C01810=1051.567,302.793,393.168,172.665,38.135,157.229
C01811=1051.561,302.545,393.201,172.661,38.131,157.228
C01812=1051.554,302.298,393.234,172.658,38.128,157.227
C01813=1051.547,302.050,393.266,172.655,38.124,157.226
C01814=1051.541,301.803,393.299,172.651,38.120,157.225
C01815=1051.534,301.555,393.332,172.648,38.117,157.225
C01816=1051.528,301.307,393.364,172.644,38.114,157.224
C01817=1051.521,301.059,393.397,172.641,38.110,157.223
C01818=1051.515,300.812,393.430,172.638,38.106,157.222
C01819=1051.508,300.565,393.462,172.634,38.103,157.221
C01820=1051.501,300.316,393.495,172.631,38.099,157.220
C01821=1051.495,300.069,393.528,172.628,38.096,157.220
C01822=1051.489,299.820,393.560,172.624,38.093,157.219
C01823=1051.483,299.573,393.593,172.621,38.089,157.218
C01824=1051.476,299.326,393.625,172.618,38.085,157.217
C01825=1051.469,299.078,393.658,172.614,38.082,157.216
C01826=1051.463,298.830,393.690,172.611,38.078,157.215
C01827=1051.457,298.582,393.722,172.608,38.075,157.215
C01828=1051.450,298.334,393.755,172.604,38.072,157.214
C01829=1051.443,298.087,393.788,172.601,38.068,157.213
C01830=1051.437,297.838,393.820,172.598,38.065,157.212
C01831=1051.431,297.591,393.852,172.595,38.061,157.211
C01832=1051.425,297.343,393.885,172.591,38.057,157.210
C01833=1051.419,297.095,393.917,172.587,38.054,157.210
C01834=1051.412,296.848,393.949,172.585,38.051,157.209
C01835=1051.405,296.600,393.982,172.581,38.047,157.208
C01836=1051.399,296.352,394.014,172.578,38.044,157.207
C01837=1051.392,296.105,394.046,172.575,38.040,157.206
C01838=1051.386,295.856,394.078,172.571,38.037,157.205
C01839=1051.379,295.609,394.110,172.569,38.033,157.205
C01840=1051.373,295.361,394.142,172.565,38.030,157.204
C01841=1051.366,295.114,394.175,172.561,38.027,157.203
C01842=1051.360,294.865,394.207,172.559,38.023,157.202
C01843=1051.353,294.617,394.239,172.555,38.020,157.201
C01844=1051.347,294.369,394.271,172.552,38.016,157.201
C01845=1051.340,294.122,394.303,172.549,38.013,157.200
C01846=1051.334,293.874,394.335,172.545,38.010,157.199
C01847=1051.327,293.626,394.367,172.542,38.006,157.198
C01848=1051.320,293.379,394.399,172.539,38.003,157.197
C01849=1051.314,293.130,394.431,172.536,37.999,157.197
C01850=1051.307,292.882,394.462,172.533,37.996,157.196
C01851=1051.300,292.635,394.494,172.529,37.993,157.195
C01852=1051.294,292.387,394.526,172.526,37.990,157.194
C01853=1051.287,292.139,394.558,172.523,37.986,157.193
C01854=1051.281,291.891,394.590,172.520,37.983,157.193
C01855=1051.274,291.644,394.622,172.516,37.979,157.192
C01856=1051.268,291.396,394.654,172.513,37.976,157.191
C01857=1051.262,291.147,394.686,172.510,37.972,157.190
C01858=1051.255,290.882,394.720,172.506,37.969,157.189
C01859=1051.247,290.617,394.753,172.503,37.966,157.189
C01860=1051.240,290.351,394.787,172.500,37.962,157.188
C01861=1051.233,290.085,394.821,172.496,37.958,157.187
C01862=1051.226,289.838,394.853,172.493,37.955,157.186
C01863=1051.220,289.589,394.885,172.490,37.952,157.185
C01864=1051.213,289.341,394.917,172.487,37.949,157.185
C01865=1051.207,289.094,394.948,172.484,37.945,157.184
C01866=1051.201,288.846,394.980,172.480,37.942,157.183
C01867=1051.195,288.598,395.011,172.478,37.938,157.182
C01868=1051.188,288.350,395.043,172.474,37.935,157.181
C01869=1051.181,288.102,395.074,172.471,37.932,157.181
C01870=1051.175,287.854,395.106,172.468,37.929,157.180
C01871=1051.168,287.606,395.138,172.465,37.925,157.179
C01872=1051.162,287.358,395.169,172.462,37.922,157.178
C01873=1051.155,287.110,395.200,172.459,37.919,157.178
C01874=1051.148,286.863,395.232,172.455,37.915,157.177
C01875=1051.142,286.615,395.263,172.453,37.912,157.176
C01876=1051.135,286.367,395.294,172.449,37.909,157.175
C01877=1051.129,286.120,395.326,172.447,37.906,157.175
C01878=1051.122,285.871,395.356,172.443,37.902,157.174
C01879=1051.116,285.623,395.388,172.440,37.899,157.173
C01880=1051.109,285.375,395.419,172.437,37.896,157.172
C01881=1051.102,285.127,395.451,172.434,37.892,157.171
C01882=1051.095,284.879,395.482,172.431,37.889,157.171
C01883=1051.089,284.632,395.514,172.428,37.886,157.170
C01884=1051.083,284.384,395.544,172.424,37.883,157.169
C01885=1051.076,284.136,395.575,172.422,37.879,157.168
C01886=1051.069,283.888,395.607,172.418,37.876,157.168
C01887=1051.063,283.640,395.639,172.416,37.873,157.167
C01888=1051.057,283.391,395.670,172.412,37.870,157.166
C01889=1051.051,283.144,395.701,172.409,37.866,157.165
C01890=1051.044,282.896,395.732,172.406,37.863,157.165
C01891=1051.038,282.648,395.763,172.403,37.860,157.164
C01892=1051.031,282.400,395.794,172.401,37.856,157.163
C01893=1051.024,282.152,395.826,172.397,37.853,157.162
C01894=1051.018,281.904,395.856,172.394,37.850,157.162
C01895=1051.012,281.656,395.887,172.391,37.847,157.161
C01896=1051.005,281.408,395.919,172.388,37.844,157.160
C01897=1050.999,281.160,395.950,172.385,37.840,157.159
C01898=1050.992,280.912,395.981,172.382,37.837,157.159
C01899=1050.986,280.664,396.011,172.379,37.833,157.158
C01900=1050.979,280.416,396.043,172.376,37.830,157.157
C01901=1050.973,280.169,396.074,172.373,37.827,157.156
C01902=1050.967,279.920,396.105,172.370,37.824,157.155
C01903=1050.960,279.672,396.136,172.367,37.821,157.155
C01904=1050.954,279.424,396.166,172.365,37.817,157.154
C01905=1050.947,279.177,396.197,172.361,37.814,157.153
C01906=1050.940,278.928,396.228,172.358,37.811,157.153
C01907=1050.934,278.680,396.259,172.355,37.807,157.152
C01908=1050.928,278.433,396.290,172.352,37.805,157.151
C01909=1050.921,278.184,396.320,172.349,37.801,157.150
C01910=1050.914,277.937,396.351,172.346,37.798,157.150
C01911=1050.908,277.689,396.382,172.344,37.795,157.149
C01912=1050.902,277.440,396.412,172.340,37.791,157.148
C01913=1050.895,277.192,396.444,172.337,37.788,157.147
C01914=1050.889,276.938,396.475,172.335,37.785,157.147
C01915=1050.882,276.684,396.507,172.331,37.782,157.146
C01916=1050.875,276.430,396.538,172.329,37.779,157.145
C01917=1050.868,276.175,396.569,172.325,37.775,157.144
C01918=1050.862,275.927,396.600,172.322,37.772,157.144
C01919=1050.855,275.679,396.630,172.320,37.769,157.143
C01920=1050.849,275.432,396.661,172.316,37.765,157.142
C01921=1050.843,275.184,396.692,172.314,37.762,157.141
C01922=1050.836,274.935,396.722,172.310,37.759,157.141
C01923=1050.830,274.688,396.752,172.308,37.756,157.140
C01924=1050.823,274.439,396.783,172.305,37.753,157.139
C01925=1050.816,274.191,396.814,172.302,37.750,157.138
C01926=1050.810,273.944,396.844,172.299,37.746,157.138
C01927=1050.803,273.695,396.875,172.296,37.743,157.137
C01928=1050.798,273.447,396.905,172.293,37.740,157.136
C01929=1050.791,273.199,396.935,172.290,37.737,157.135
C01930=1050.785,272.951,396.966,172.288,37.734,157.135
C01931=1050.778,272.703,396.996,172.284,37.730,157.134
C01932=1050.771,272.454,397.026,172.282,37.727,157.133
C01933=1050.765,272.207,397.057,172.279,37.724,157.133
C01934=1050.759,271.959,397.088,172.276,37.721,157.132
C01935=1050.752,271.711,397.118,172.273,37.717,157.131
C01936=1050.746,271.463,397.149,172.270,37.715,157.130
C01937=1050.739,271.215,397.178,172.268,37.711,157.130
C01938=1050.733,270.967,397.209,172.264,37.708,157.129
C01939=1050.726,270.719,397.238,172.262,37.705,157.128
C01940=1050.720,270.470,397.269,172.259,37.702,157.128
C01941=1050.713,270.222,397.299,172.256,37.698,157.127
C01942=1050.707,269.974,397.329,172.253,37.695,157.126
C01943=1050.700,269.726,397.360,172.250,37.692,157.125
C01944=1050.694,269.478,397.390,172.248,37.689,157.125
C01945=1050.687,269.230,397.420,172.244,37.686,157.124
C01946=1050.681,268.982,397.450,172.242,37.683,157.123
C01947=1050.674,268.734,397.480,172.239,37.680,157.123
C01948=1050.668,268.486,397.511,172.237,37.676,157.122
C01949=1050.662,268.238,397.540,172.233,37.673,157.121
C01950=1050.655,267.989,397.571,172.231,37.670,157.120
C01951=1050.649,267.742,397.600,172.228,37.667,157.120
C01952=1050.642,267.493,397.630,172.225,37.664,157.119
C01953=1050.636,267.245,397.660,172.222,37.661,157.118
C01954=1050.629,266.997,397.690,172.220,37.658,157.117
C01955=1050.622,266.749,397.720,172.217,37.654,157.117
C01956=1050.616,266.501,397.751,172.213,37.651,157.116
C01957=1050.610,266.253,397.780,172.211,37.648,157.115
C01958=1050.603,266.004,397.810,172.208,37.645,157.115
C01959=1050.597,265.757,397.840,172.206,37.642,157.114
C01960=1050.590,265.508,397.870,172.203,37.639,157.113
C01961=1050.584,265.260,397.900,172.200,37.636,157.112
C01962=1050.578,265.012,397.930,172.197,37.632,157.112
C01963=1050.571,264.764,397.959,172.195,37.629,157.111
C01964=1050.565,264.516,397.989,172.192,37.626,157.110
C01965=1050.558,264.268,398.020,172.189,37.623,157.110
C01966=1050.552,264.019,398.049,172.186,37.619,157.109
C01967=1050.546,263.772,398.079,172.183,37.617,157.108
C01968=1050.539,263.523,398.108,172.181,37.614,157.108
C01969=1050.532,263.275,398.138,172.178,37.610,157.107
C01970=1050.526,263.025,398.168,172.175,37.607,157.106
C01971=1050.520,262.776,398.198,172.172,37.604,157.105
C01972=1050.513,262.526,398.228,172.170,37.601,157.105
C01973=1050.507,262.275,398.258,172.167,37.598,157.104
C01974=1050.500,262.026,398.287,172.165,37.594,157.103
C01975=1050.493,261.779,398.317,172.161,37.592,157.103
C01976=1050.487,261.531,398.346,172.159,37.589,157.102
C01977=1050.479,261.283,398.376,172.156,37.586,157.101
C01978=1050.473,261.035,398.405,172.154,37.582,157.100
C01979=1050.466,260.786,398.434,172.150,37.579,157.100
C01980=1050.459,260.538,398.464,172.148,37.576,157.099
C01981=1050.453,260.290,398.493,172.145,37.573,157.098
C01982=1050.446,260.041,398.522,172.143,37.570,157.098
C01983=1050.440,259.794,398.552,172.140,37.567,157.097
C01984=1050.434,259.546,398.581,172.138,37.564,157.096
C01985=1050.427,259.297,398.610,172.134,37.561,157.096
C01986=1050.420,259.049,398.639,172.132,37.558,157.095
C01987=1050.414,258.801,398.669,172.129,37.555,157.094
C01988=1050.407,258.553,398.699,172.127,37.552,157.094
C01989=1050.401,258.304,398.728,172.124,37.548,157.093
C01990=1050.395,258.056,398.757,172.122,37.546,157.092
C01991=1050.387,257.808,398.787,172.118,37.543,157.092
C01992=1050.381,257.560,398.816,172.115,37.539,157.091
C01993=1050.375,257.312,398.845,172.113,37.536,157.090
C01994=1050.368,257.063,398.874,172.111,37.533,157.089
C01995=1050.362,256.815,398.903,172.108,37.530,157.089
C01996=1050.356,256.567,398.932,172.105,37.527,157.088
C01997=1050.349,256.319,398.962,172.103,37.524,157.087
C01998=1050.342,256.070,398.992,172.099,37.521,157.087
C01999=1050.336,255.822,399.021,172.097,37.518,157.086
C02000=1050.329,255.574,399.049,172.094,37.515,157.085
C02001=1050.323,255.326,399.078,172.092,37.512,157.085
C02002=1050.316,255.077,399.107,172.089,37.508,157.084
C02003=1050.310,254.829,399.136,172.087,37.505,157.083
C02004=1050.303,254.581,399.166,172.084,37.502,157.083
C02005=1050.297,254.333,399.195,172.082,37.499,157.082
C02006=1050.291,254.085,399.224,172.079,37.496,157.081
C02007=1050.284,253.836,399.253,172.077,37.493,157.080
C02008=1050.278,253.588,399.282,172.073,37.490,157.080
C02009=1050.271,253.340,399.311,172.071,37.487,157.079
C02010=1050.265,253.092,399.340,172.068,37.484,157.078
C02011=1050.258,252.844,399.369,172.066,37.480,157.078
C02012=1050.251,252.595,399.398,172.063,37.477,157.077
C02013=1050.245,252.347,399.427,172.061,37.474,157.076
C02014=1050.239,252.099,399.456,172.058,37.471,157.076
C02015=1050.233,251.851,399.485,172.056,37.468,157.075
C02016=1050.226,251.602,399.514,172.053,37.465,157.074
C02017=1050.220,251.354,399.543,172.051,37.461,157.073
C02018=1050.214,251.106,399.572,172.048,37.458,157.073
C02019=1050.208,250.858,399.601,172.046,37.456,157.072
C02020=1050.201,250.609,399.630,172.043,37.452,157.071
C02021=1050.194,250.361,399.658,172.041,37.449,157.071
C02022=1050.188,250.113,399.687,172.038,37.446,157.070
C02023=1050.182,249.865,399.716,172.036,37.443,157.069
C02024=1050.175,249.616,399.746,172.033,37.440,157.069
C02025=1050.169,249.368,399.775,172.031,37.437,157.068
C02026=1050.162,249.116,399.804,172.028,37.433,157.067
C02027=1050.156,248.865,399.833,172.026,37.430,157.067
C02028=1050.150,248.613,399.862,172.022,37.427,157.066
C02029=1050.144,248.362,399.891,172.020,37.424,157.065
C02030=1050.138,248.114,399.919,172.017,37.420,157.064
C02031=1050.131,247.865,399.948,172.015,37.417,157.064
C02032=1050.125,247.617,399.977,172.012,37.415,157.063
C02033=1050.119,247.369,400.007,172.010,37.411,157.062
C02034=1050.112,247.121,400.034,172.007,37.408,157.062
C02035=1050.106,246.873,400.063,172.005,37.405,157.061
C02036=1050.100,246.625,400.092,172.003,37.402,157.060
C02037=1050.094,246.376,400.121,172.001,37.399,157.060
C02038=1050.087,246.128,400.150,171.998,37.395,157.059
C02039=1050.081,245.879,400.179,171.996,37.392,157.058
C02040=1050.075,245.631,400.206,171.993,37.389,157.057
C02041=1050.068,245.382,400.236,171.991,37.386,157.057
C02042=1050.062,245.133,400.264,171.988,37.383,157.056
C02043=1050.055,244.886,400.293,171.986,37.380,157.055
C02044=1050.049,244.637,400.321,171.983,37.376,157.055
C02045=1050.042,244.389,400.349,171.981,37.373,157.054
C02046=1050.036,244.141,400.378,171.978,37.370,157.053
C02047=1050.030,243.892,400.407,171.976,37.367,157.053
C02048=1050.023,243.644,400.435,171.973,37.364,157.052
C02049=1050.017,243.396,400.464,171.971,37.361,157.051
C02050=1050.011,243.148,400.491,171.968,37.358,157.051
C02051=1050.004,242.900,400.520,171.966,37.355,157.050
C02052=1049.998,242.651,400.548,171.963,37.352,157.049
C02053=1049.991,242.403,400.577,171.961,37.349,157.049
C02054=1049.986,242.154,400.605,171.958,37.345,157.048
C02055=1049.979,241.907,400.633,171.956,37.342,157.047
C02056=1049.973,241.658,400.662,171.953,37.339,157.047
C02057=1049.966,241.409,400.690,171.951,37.336,157.046
C02058=1049.960,241.161,400.719,171.948,37.333,157.045
C02059=1049.953,240.913,400.746,171.946,37.330,157.044
C02060=1049.946,240.664,400.774,171.943,37.327,157.044
C02061=1049.940,240.416,400.803,171.942,37.323,157.043
C02062=1049.933,240.168,400.831,171.939,37.320,157.042
C02063=1049.927,239.919,400.859,171.937,37.317,157.042
C02064=1049.921,239.671,400.887,171.934,37.314,157.041
C02065=1049.914,239.423,400.915,171.932,37.311,157.040
C02066=1049.908,239.174,400.944,171.929,37.308,157.040
C02067=1049.901,238.926,400.971,171.927,37.305,157.039
C02068=1049.894,238.677,400.999,171.924,37.302,157.038
C02069=1049.888,238.429,401.028,171.922,37.299,157.038
C02070=1049.882,238.181,401.056,171.919,37.296,157.037
C02071=1049.875,237.933,401.083,171.917,37.293,157.036
C02072=1049.869,237.684,401.112,171.915,37.290,157.036
C02073=1049.863,237.436,401.139,171.913,37.286,157.035
C02074=1049.856,237.187,401.167,171.911,37.283,157.034
C02075=1049.849,236.939,401.195,171.908,37.280,157.034
C02076=1049.843,236.691,401.224,171.906,37.277,157.033
C02077=1049.837,236.442,401.252,171.903,37.274,157.032
C02078=1049.830,236.194,401.279,171.901,37.271,157.032
C02079=1049.824,235.946,401.307,171.898,37.268,157.031
C02080=1049.818,235.697,401.335,171.896,37.265,157.030
C02081=1049.811,235.449,401.363,171.893,37.261,157.030
C02082=1049.805,235.191,401.392,171.892,37.258,157.029
C02083=1049.797,234.934,401.421,171.889,37.255,157.028
C02084=1049.792,234.677,401.450,171.887,37.252,157.027
C02085=1049.784,234.419,401.478,171.884,37.248,157.027
C02086=1049.778,234.171,401.507,171.882,37.245,157.026
C02087=1049.772,233.922,401.534,171.879,37.242,157.025
C02088=1049.765,233.674,401.562,171.877,37.239,157.025
C02089=1049.759,233.426,401.589,171.874,37.236,157.024
C02090=1049.753,233.177,401.618,171.873,37.233,157.023
C02091=1049.746,232.929,401.645,171.870,37.230,157.023
C02092=1049.740,232.680,401.673,171.868,37.226,157.022
C02093=1049.733,232.432,401.701,171.865,37.224,157.021
C02094=1049.727,232.184,401.728,171.863,37.221,157.021
C02095=1049.721,231.935,401.756,171.860,37.217,157.020
C02096=1049.715,231.686,401.784,171.859,37.214,157.019
C02097=1049.708,231.438,401.811,171.857,37.211,157.019
C02098=1049.702,231.190,401.839,171.854,37.208,157.018
C02099=1049.695,230.942,401.866,171.852,37.205,157.017
C02100=1049.689,230.693,401.894,171.849,37.202,157.017
C02101=1049.682,230.445,401.922,171.847,37.199,157.016
C02102=1049.676,230.197,401.949,171.845,37.195,157.015
C02103=1049.669,229.948,401.976,171.843,37.192,157.015
C02104=1049.663,229.699,402.005,171.840,37.189,157.014
C02105=1049.657,229.451,402.032,171.838,37.186,157.013
C02106=1049.651,229.203,402.060,171.835,37.183,157.013
C02107=1049.644,228.954,402.087,171.834,37.180,157.012
C02108=1049.638,228.706,402.114,171.831,37.177,157.011
C02109=1049.631,228.457,402.142,171.829,37.173,157.010
C02110=1049.625,228.209,402.169,171.826,37.170,157.010
C02111=1049.618,227.961,402.196,171.824,37.167,157.009
C02112=1049.611,227.712,402.224,171.823,37.164,157.009
C02113=1049.605,227.463,402.251,171.820,37.161,157.008
C02114=1049.599,227.216,402.278,171.818,37.158,157.007
C02115=1049.592,226.967,402.306,171.815,37.155,157.007
C02116=1049.586,226.718,402.333,171.814,37.152,157.006
C02117=1049.579,226.470,402.361,171.811,37.148,157.005
C02118=1049.573,226.221,402.387,171.809,37.145,157.004
C02119=1049.566,225.973,402.415,171.806,37.142,157.004
C02120=1049.559,225.725,402.442,171.804,37.139,157.003
C02121=1049.553,225.476,402.469,171.802,37.136,157.002
C02122=1049.547,225.228,402.496,171.800,37.133,157.002
C02123=1049.540,224.979,402.523,171.797,37.130,157.001
C02124=1049.534,224.731,402.551,171.795,37.126,157.000
C02125=1049.528,224.482,402.578,171.794,37.123,157.000
C02126=1049.521,224.234,402.606,171.791,37.120,156.999
C02127=1049.515,223.985,402.632,171.789,37.117,156.999
C02128=1049.508,223.737,402.659,171.786,37.114,156.998
C02129=1049.502,223.489,402.686,171.785,37.111,156.997
C02130=1049.495,223.240,402.714,171.782,37.108,156.996
C02131=1049.489,222.991,402.741,171.780,37.104,156.996
C02132=1049.483,222.744,402.768,171.778,37.101,156.995
C02133=1049.477,222.494,402.795,171.776,37.098,156.994
C02134=1049.470,222.246,402.823,171.773,37.095,156.994
C02135=1049.463,221.998,402.849,171.771,37.092,156.993
C02136=1049.457,221.750,402.877,171.770,37.089,156.992
C02137=1049.451,221.501,402.903,171.767,37.085,156.992
C02138=1049.445,221.236,402.932,171.765,37.082,156.991
C02139=1049.437,220.971,402.961,171.762,37.079,156.990
C02140=1049.430,220.706,402.989,171.761,37.075,156.990
C02141=1049.424,220.441,403.019,171.758,37.072,156.989
C02142=1049.417,220.192,403.046,171.756,37.069,156.988
C02143=1049.411,219.944,403.072,171.753,37.066,156.987
C02144=1049.404,219.696,403.099,171.752,37.063,156.987
C02145=1049.398,219.447,403.126,171.749,37.059,156.986
C02146=1049.391,219.199,403.153,171.747,37.056,156.985
C02147=1049.385,218.950,403.180,171.744,37.053,156.985
C02148=1049.378,218.702,403.206,171.743,37.050,156.984
C02149=1049.371,218.453,403.233,171.740,37.047,156.983
C02150=1049.365,218.205,403.259,171.738,37.044,156.983
C02151=1049.359,217.956,403.286,171.737,37.041,156.982
C02152=1049.352,217.708,403.314,171.734,37.038,156.982
C02153=1049.345,217.460,403.340,171.732,37.034,156.981
C02154=1049.339,217.211,403.367,171.730,37.031,156.980
C02155=1049.333,216.962,403.393,171.728,37.028,156.979
C02156=1049.326,216.713,403.420,171.725,37.024,156.979
C02157=1049.320,216.465,403.447,171.724,37.021,156.978
C02158=1049.313,216.217,403.474,171.721,37.018,156.977
C02159=1049.307,215.969,403.501,171.719,37.015,156.977
C02160=1049.300,215.720,403.527,171.717,37.012,156.976
C02161=1049.294,215.471,403.554,171.715,37.009,156.975
C02162=1049.287,215.223,403.580,171.713,37.005,156.975
C02163=1049.281,214.974,403.607,171.711,37.002,156.974
C02164=1049.275,214.725,403.634,171.709,36.999,156.973
C02165=1049.269,214.477,403.660,171.707,36.996,156.973
C02166=1049.262,214.228,403.687,171.705,36.993,156.972
C02167=1049.256,213.980,403.713,171.702,36.989,156.971
C02168=1049.250,213.732,403.740,171.701,36.986,156.971
C02169=1049.243,213.483,403.766,171.698,36.983,156.970
C02170=1049.237,213.235,403.793,171.696,36.980,156.969
C02171=1049.230,212.986,403.819,171.695,36.977,156.969
C02172=1049.224,212.738,403.846,171.692,36.974,156.968
C02173=1049.217,212.489,403.872,171.691,36.970,156.967
C02174=1049.211,212.240,403.899,171.688,36.967,156.967
C02175=1049.204,211.992,403.925,171.686,36.964,156.966
C02176=1049.198,211.743,403.952,171.684,36.961,156.965
C02177=1049.192,211.495,403.978,171.682,36.958,156.965
C02178=1049.185,211.246,404.005,171.680,36.954,156.964
C02179=1049.179,210.998,404.031,171.678,36.951,156.963
C02180=1049.172,210.749,404.057,171.676,36.948,156.963
C02181=1049.166,210.501,404.084,171.674,36.944,156.962
C02182=1049.159,210.252,404.110,171.672,36.941,156.961
C02183=1049.153,210.004,404.137,171.670,36.938,156.960
C02184=1049.147,209.755,404.162,171.668,36.935,156.960
C02185=1049.140,209.507,404.189,171.665,36.932,156.959
C02186=1049.134,209.258,404.216,171.664,36.928,156.958
C02187=1049.127,209.009,404.242,171.661,36.925,156.958
C02188=1049.120,208.761,404.268,171.660,36.922,156.957
C02189=1049.114,208.513,404.293,171.657,36.919,156.956
C02190=1049.108,208.264,404.320,171.656,36.916,156.956
C02191=1049.101,208.016,404.346,171.654,36.912,156.955
C02192=1049.095,207.768,404.372,171.651,36.909,156.954
C02193=1049.088,207.518,404.399,171.650,36.906,156.954
C02194=1049.082,207.258,404.426,171.647,36.903,156.953
C02195=1049.075,207.000,404.453,171.646,36.899,156.952
C02196=1049.068,206.740,404.481,171.643,36.896,156.952
C02197=1049.061,206.481,404.508,171.641,36.892,156.951
C02198=1049.035,205.428,404.614,171.404,36.795,156.930
C02199=1049.029,205.180,404.639,171.402,36.792,156.929
C02200=1049.023,204.932,404.664,171.400,36.790,156.929
C02201=1049.017,204.683,404.689,171.396,36.788,156.928
C02202=1049.011,204.434,404.714,171.394,36.785,156.928
C02203=1049.005,204.185,404.739,171.392,36.783,156.927
C02204=1048.999,203.936,404.765,171.388,36.780,156.927
C02205=1048.993,203.688,404.789,171.386,36.778,156.926
C02206=1048.987,203.439,404.814,171.384,36.776,156.926
C02207=1048.981,203.190,404.839,171.382,36.773,156.925
C02208=1048.974,202.942,404.864,171.378,36.771,156.925
C02209=1048.969,202.694,404.888,171.376,36.768,156.924
C02210=1048.963,202.445,404.914,171.374,36.766,156.924
C02211=1048.957,202.196,404.938,171.370,36.763,156.923
C02212=1048.951,201.947,404.964,171.368,36.761,156.923
C02213=1048.945,201.699,404.989,171.366,36.759,156.923
C02214=1048.939,201.450,405.013,171.363,36.756,156.922
C02215=1048.932,201.201,405.038,171.360,36.754,156.922
C02216=1048.926,200.952,405.063,171.358,36.752,156.921
C02217=1048.921,200.704,405.088,171.355,36.750,156.921
C02218=1048.914,200.455,405.112,171.352,36.747,156.920
C02219=1048.908,200.206,405.137,171.350,36.745,156.920
C02220=1048.902,199.957,405.162,171.348,36.742,156.919
C02221=1048.895,199.709,405.186,171.345,36.741,156.919
C02222=1048.890,199.460,405.211,171.342,36.738,156.918
C02223=1048.883,199.211,405.235,171.340,36.736,156.918
C02224=1048.877,198.963,405.260,171.337,36.733,156.917
C02225=1048.871,198.714,405.284,171.335,36.731,156.917
C02226=1048.865,198.466,405.309,171.332,36.729,156.916
C02227=1048.859,198.216,405.334,171.329,36.727,156.916
C02228=1048.852,197.968,405.358,171.327,36.724,156.915
C02229=1048.847,197.719,405.383,171.325,36.722,156.915
C02230=1048.840,197.470,405.407,171.322,36.720,156.915
C02231=1048.834,197.222,405.432,171.319,36.718,156.914
C02232=1048.828,196.973,405.456,171.317,36.715,156.914
C02233=1048.822,196.724,405.480,171.315,36.713,156.913
C02234=1048.816,196.475,405.506,171.311,36.711,156.913
C02235=1048.809,196.227,405.529,171.309,36.709,156.912
C02236=1048.804,195.978,405.554,171.307,36.706,156.912
C02237=1048.797,195.729,405.578,171.305,36.704,156.911
C02238=1048.791,195.481,405.603,171.301,36.702,156.911
C02239=1048.785,195.232,405.627,171.299,36.700,156.910
C02240=1048.779,194.983,405.652,171.297,36.697,156.910
C02241=1048.774,194.734,405.676,171.294,36.695,156.909
C02242=1048.767,194.486,405.701,171.292,36.693,156.909
C02243=1048.761,194.237,405.725,171.289,36.690,156.908
C02244=1048.755,193.988,405.749,171.287,36.688,156.908
C02245=1048.749,193.739,405.773,171.284,36.686,156.908
C02246=1048.742,193.491,405.798,171.282,36.684,156.907
C02247=1048.736,193.242,405.822,171.279,36.681,156.907
C02248=1048.730,192.994,405.846,171.276,36.679,156.906
C02249=1048.725,192.744,405.871,171.274,36.677,156.906
C02250=1048.719,192.496,405.894,171.272,36.675,156.905
C02251=1048.713,192.247,405.919,171.270,36.672,156.905
C02252=1048.706,191.998,405.943,171.267,36.670,156.904
C02253=1048.700,191.750,405.968,171.264,36.668,156.904
C02254=1048.694,191.501,405.992,171.262,36.666,156.903
C02255=1048.688,191.252,406.016,171.259,36.663,156.903
C02256=1048.683,191.003,406.041,171.257,36.661,156.903
C02257=1048.676,190.755,406.065,171.255,36.659,156.902
C02258=1048.671,190.505,406.089,171.253,36.657,156.902
C02259=1048.664,190.221,406.116,171.249,36.654,156.901
C02260=1048.657,189.937,406.144,171.247,36.652,156.901
C02261=1048.650,189.652,406.172,171.244,36.649,156.900
C02262=1048.643,189.369,406.199,171.241,36.647,156.900
C02263=1048.637,189.119,406.224,171.239,36.644,156.899
C02264=1048.631,188.871,406.248,171.236,36.642,156.899
C02265=1048.625,188.622,406.272,171.233,36.640,156.898
C02266=1048.619,188.374,406.296,171.231,36.638,156.898
C02267=1048.613,188.124,406.321,171.229,36.635,156.897
C02268=1048.607,187.876,406.344,171.227,36.633,156.897
C02269=1048.602,187.627,406.368,171.224,36.631,156.896
C02270=1048.596,187.378,406.392,171.222,36.629,156.896
C02271=1048.590,187.129,406.416,171.219,36.627,156.896
C02272=1048.584,186.880,406.440,171.217,36.624,156.895
C02273=1048.578,186.632,406.464,171.214,36.622,156.895
C02274=1048.572,186.383,406.488,171.212,36.620,156.894
C02275=1048.566,186.134,406.513,171.210,36.618,156.894
C02276=1048.560,185.886,406.536,171.207,36.615,156.893
C02277=1048.554,185.637,406.560,171.205,36.613,156.893
C02278=1048.548,185.388,406.585,171.203,36.611,156.892
C02279=1048.543,185.139,406.607,171.201,36.609,156.892
C02280=1048.537,184.890,406.632,171.197,36.607,156.891
C02281=1048.531,184.642,406.656,171.195,36.604,156.891
C02282=1048.525,184.393,406.680,171.193,36.602,156.890
C02283=1048.519,184.144,406.704,171.190,36.600,156.890
C02284=1048.514,183.895,406.728,171.188,36.598,156.890
C02285=1048.507,183.646,406.752,171.186,36.596,156.889
C02286=1048.501,183.398,406.775,171.184,36.594,156.889
C02287=1048.494,183.148,406.798,171.181,36.592,156.888
C02288=1048.488,182.900,406.822,171.179,36.590,156.888
C02289=1048.481,182.651,406.846,171.176,36.587,156.888
C02290=1048.476,182.402,406.869,171.174,36.585,156.887
C02291=1048.469,182.153,406.893,171.171,36.584,156.887
C02292=1048.463,181.904,406.916,171.169,36.581,156.886
C02293=1048.457,181.656,406.939,171.167,36.579,156.886
C02294=1048.451,181.407,406.963,171.165,36.578,156.886
C02295=1048.445,181.158,406.986,171.162,36.575,156.885
C02296=1048.438,180.909,407.010,171.160,36.573,156.885
C02297=1048.432,180.660,407.033,171.157,36.571,156.884
C02298=1048.426,180.411,407.057,171.155,36.570,156.884
C02299=1048.420,180.163,407.080,171.152,36.567,156.883
C02300=1048.414,179.914,407.104,171.150,36.565,156.883
C02301=1048.408,179.665,407.127,171.148,36.564,156.883
C02302=1048.401,179.417,407.150,171.146,36.561,156.882
C02303=1048.395,179.168,407.173,171.144,36.559,156.882
C02304=1048.389,178.919,407.197,171.141,36.557,156.882
C02305=1048.383,178.670,407.220,171.139,36.555,156.881
C02306=1048.376,178.421,407.244,171.137,36.553,156.881
C02307=1048.371,178.172,407.267,171.134,36.551,156.880
C02308=1048.364,177.924,407.291,171.131,36.549,156.880
C02309=1048.358,177.674,407.314,171.129,36.547,156.879
C02310=1048.352,177.426,407.338,171.127,36.545,156.879
C02311=1048.346,177.177,407.361,171.125,36.543,156.879
C02312=1048.340,176.927,407.384,171.122,36.541,156.878
C02313=1048.333,176.679,407.407,171.120,36.539,156.878
C02314=1048.328,176.431,407.430,171.118,36.537,156.877
C02315=1048.321,176.182,407.454,171.116,36.535,156.877
C02316=1048.315,175.933,407.477,171.113,36.533,156.877
C02317=1048.309,175.684,407.500,171.111,36.531,156.876
C02318=1048.303,175.436,407.524,171.109,36.529,156.876
C02319=1048.297,175.186,407.547,171.107,36.527,156.875
C02320=1048.291,174.937,407.570,171.104,36.525,156.875
C02321=1048.285,174.689,407.593,171.102,36.523,156.875
C02322=1048.279,174.440,407.616,171.100,36.521,156.874
C02323=1048.272,174.155,407.643,171.097,36.518,156.874
C02324=1048.264,173.870,407.669,171.094,36.517,156.873
C02325=1048.258,173.585,407.696,171.092,36.514,156.873
C02326=1048.251,173.300,407.722,171.089,36.512,156.872
C02327=1048.245,173.052,407.745,171.087,36.510,156.872
C02328=1048.239,172.803,407.768,171.084,36.508,156.872
C02329=1048.233,172.554,407.791,171.082,36.506,156.871
C02330=1048.227,172.305,407.814,171.080,36.504,156.871
C02331=1048.221,172.056,407.838,171.078,36.502,156.870
C02332=1048.215,171.807,407.861,171.075,36.499,156.870
C02333=1048.209,171.558,407.884,171.073,36.498,156.870
C02334=1048.203,171.310,407.906,171.071,36.496,156.869
C02335=1048.197,171.060,407.930,171.069,36.494,156.869
C02336=1048.190,170.812,407.953,171.066,36.492,156.868
C02337=1048.185,170.563,407.976,171.064,36.490,156.868
C02338=1048.179,170.314,407.999,171.062,36.488,156.868
C02339=1048.173,170.065,408.022,171.060,36.485,156.867
C02340=1048.167,169.817,408.045,171.057,36.484,156.867
C02341=1048.161,169.568,408.067,171.055,36.482,156.866
C02342=1048.155,169.318,408.091,171.053,36.480,156.866
C02343=1048.149,169.069,408.114,171.051,36.477,156.866
C02344=1048.143,168.821,408.137,171.049,36.476,156.865
C02345=1048.137,168.572,408.160,171.046,36.474,156.865
C02346=1048.131,168.324,408.183,171.044,36.472,156.864
C02347=1048.125,168.075,408.206,171.042,36.470,156.864
C02348=1048.119,167.826,408.229,171.040,36.468,156.864
C02349=1048.114,167.577,408.252,171.037,36.466,156.863
C02350=1048.108,167.328,408.274,171.035,36.463,156.863
C02351=1048.102,167.078,408.298,171.033,36.462,156.862
C02352=1048.095,166.830,408.320,171.031,36.460,156.862
C02353=1048.089,166.581,408.343,171.028,36.458,156.862
C02354=1048.084,166.332,408.366,171.026,36.455,156.861
C02355=1048.078,166.083,408.389,171.025,36.454,156.861
C02356=1048.072,165.834,408.412,171.023,36.452,156.860
C02357=1048.066,165.586,408.434,171.021,36.450,156.860
C02358=1048.060,165.337,408.457,171.018,36.447,156.860
C02359=1048.054,165.088,408.480,171.016,36.446,156.859
C02360=1048.048,164.839,408.503,171.014,36.444,156.859
C02361=1048.043,164.590,408.526,171.012,36.442,156.858
C02362=1048.036,164.341,408.548,171.009,36.439,156.858
C02363=1048.031,164.093,408.571,171.007,36.438,156.858
C02364=1048.025,163.843,408.594,171.005,36.436,156.857
C02365=1048.019,163.594,408.617,171.003,36.434,156.857
C02366=1048.013,163.346,408.639,171.000,36.432,156.856
C02367=1048.007,163.097,408.662,170.998,36.430,156.856
C02368=1048.001,162.848,408.685,170.996,36.428,156.856
C02369=1047.996,162.599,408.708,170.994,36.426,156.855
C02370=1047.990,162.350,408.731,170.991,36.424,156.855
C02371=1047.984,162.101,408.753,170.990,36.422,156.854
C02372=1047.978,161.852,408.775,170.988,36.420,156.854
C02373=1047.972,161.603,408.798,170.986,36.417,156.854
C02374=1047.967,161.354,408.821,170.984,36.416,156.853
C02375=1047.960,161.106,408.843,170.981,36.414,156.853
C02376=1047.954,160.857,408.866,170.979,36.412,156.853
C02377=1047.949,160.607,408.889,170.977,36.409,156.852
C02378=1047.943,160.359,408.911,170.975,36.408,156.852
C02379=1047.937,160.110,408.934,170.972,36.406,156.851
C02380=1047.931,159.860,408.956,170.970,36.404,156.851
C02381=1047.925,159.612,408.979,170.968,36.402,156.851
C02382=1047.918,159.363,409.001,170.966,36.400,156.850
C02383=1047.912,159.114,409.023,170.965,36.398,156.850
C02384=1047.907,158.865,409.045,170.962,36.396,156.850
C02385=1047.900,158.616,409.068,170.960,36.395,156.849
C02386=1047.895,158.367,409.090,170.958,36.393,156.849
C02387=1047.888,158.082,409.116,170.956,36.390,156.848
C02388=1047.881,157.796,409.141,170.952,36.388,156.848
C02389=1047.873,157.511,409.167,170.950,36.387,156.848
C02390=1047.867,157.226,409.192,170.948,36.384,156.847
C02391=1047.860,156.978,409.214,170.946,36.382,156.847
C02392=1047.855,156.728,409.237,170.944,36.380,156.846
C02393=1047.848,156.480,409.259,170.941,36.379,156.846
C02394=1047.843,156.230,409.281,170.939,36.377,156.846
C02395=1047.836,155.981,409.304,170.937,36.375,156.845
C02396=1047.830,155.732,409.325,170.936,36.373,156.845
C02397=1047.824,155.483,409.348,170.934,36.371,156.845
C02398=1047.818,155.234,409.370,170.931,36.369,156.844
C02399=1047.812,154.986,409.392,170.929,36.368,156.844
C02400=1047.807,154.737,409.414,170.927,36.366,156.843
C02401=1047.800,154.488,409.436,170.925,36.364,156.843
C02402=1047.794,154.239,409.458,170.923,36.362,156.843
C02403=1047.788,153.990,409.480,170.920,36.360,156.842
C02404=1047.782,153.741,409.503,170.918,36.358,156.842
C02405=1047.776,153.492,409.525,170.917,36.356,156.842
C02406=1047.770,153.243,409.547,170.915,36.355,156.841
C02407=1047.764,152.994,409.568,170.912,36.353,156.841
C02408=1047.758,152.745,409.591,170.910,36.351,156.841
C02409=1047.752,152.496,409.613,170.908,36.349,156.840
C02410=1047.745,152.247,409.635,170.906,36.347,156.840
C02411=1047.740,151.999,409.656,170.904,36.345,156.839
C02412=1047.734,151.749,409.678,170.901,36.344,156.839
C02413=1047.728,151.501,409.701,170.899,36.342,156.839
C02414=1047.722,151.251,409.723,170.898,36.340,156.838
C02415=1047.715,151.002,409.744,170.896,36.338,156.838
C02416=1047.709,150.754,409.767,170.894,36.336,156.838
C02417=1047.704,150.504,409.789,170.891,36.334,156.837
C02418=1047.698,150.256,409.810,170.889,36.332,156.837
C02419=1047.692,150.007,409.832,170.887,36.331,156.837
C02420=1047.685,149.758,409.854,170.885,36.329,156.836
C02421=1047.679,149.509,409.876,170.884,36.327,156.836
C02422=1047.673,149.260,409.898,170.881,36.325,156.836
C02423=1047.667,149.010,409.920,170.879,36.323,156.835
C02424=1047.662,148.762,409.942,170.877,36.321,156.835
C02425=1047.656,148.513,409.963,170.875,36.319,156.834
C02426=1047.649,148.264,409.986,170.873,36.318,156.834
C02427=1047.643,148.015,410.007,170.870,36.316,156.834
C02428=1047.637,147.766,410.029,170.869,36.314,156.833
C02429=1047.631,147.517,410.050,170.867,36.312,156.833
C02430=1047.625,147.268,410.072,170.865,36.311,156.833
C02431=1047.619,147.019,410.094,170.863,36.309,156.832
C02432=1047.612,146.770,410.116,170.860,36.307,156.832
C02433=1047.606,146.521,410.137,170.858,36.305,156.832
C02434=1047.600,146.272,410.159,170.856,36.303,156.831
C02435=1047.595,146.023,410.180,170.855,36.302,156.831
C02436=1047.588,145.774,410.202,170.853,36.300,156.831
C02437=1047.582,145.525,410.224,170.850,36.298,156.830
C02438=1047.576,145.276,410.245,170.848,36.297,156.830
C02439=1047.570,145.026,410.267,170.846,36.295,156.830
C02440=1047.564,144.779,410.289,170.844,36.293,156.829
C02441=1047.558,144.529,410.310,170.843,36.291,156.829
C02442=1047.552,144.280,410.332,170.840,36.289,156.829
C02443=1047.546,144.031,410.354,170.838,36.287,156.828
C02444=1047.539,143.782,410.375,170.836,36.285,156.828
C02445=1047.534,143.533,410.397,170.834,36.284,156.827
C02446=1047.528,143.284,410.418,170.832,36.282,156.827
C02447=1047.522,143.035,410.440,170.831,36.280,156.827
C02448=1047.515,142.786,410.462,170.828,36.279,156.827
C02449=1047.510,142.537,410.483,170.826,36.277,156.826
C02450=1047.503,142.288,410.504,170.824,36.275,156.826
C02451=1047.497,142.003,410.528,170.822,36.273,156.825
C02452=1047.489,141.717,410.553,170.819,36.271,156.825
C02453=1047.483,141.432,410.578,170.817,36.269,156.825
C02454=1047.475,141.146,410.602,170.815,36.267,156.824
C02455=1047.470,140.897,410.624,170.813,36.265,156.824
C02456=1047.464,140.648,410.645,170.811,36.263,156.824
C02457=1047.457,140.399,410.667,170.808,36.261,156.823
C02458=1047.452,140.150,410.688,170.807,36.259,156.823
C02459=1047.446,139.901,410.710,170.805,36.258,156.822
C02460=1047.439,139.652,410.731,170.803,36.256,156.822
C02461=1047.433,139.403,410.753,170.801,36.254,156.822
C02462=1047.427,139.154,410.773,170.799,36.253,156.822
C02463=1047.421,138.905,410.795,170.797,36.251,156.821
C02464=1047.415,138.655,410.816,170.795,36.249,156.821
C02465=1047.409,138.407,410.838,170.793,36.248,156.821
C02466=1047.403,138.158,410.859,170.791,36.246,156.820
C02467=1047.396,137.909,410.880,170.789,36.244,156.820
C02468=1047.391,137.660,410.901,170.787,36.242,156.819
C02469=1047.385,137.410,410.922,170.785,36.240,156.819
C02470=1047.378,137.161,410.944,170.783,36.239,156.819
C02471=1047.373,136.913,410.965,170.781,36.237,156.819
C02472=1047.366,136.664,410.986,170.779,36.235,156.818
C02473=1047.360,136.414,411.007,170.777,36.233,156.818
C02474=1047.354,136.166,411.028,170.775,36.231,156.817
C02475=1047.348,135.917,411.050,170.773,36.230,156.817
C02476=1047.342,135.667,411.071,170.771,36.228,156.817
C02477=1047.336,135.419,411.091,170.769,36.227,156.817
C02478=1047.330,135.169,411.113,170.768,36.225,156.816
C02479=1047.324,134.920,411.135,170.765,36.223,156.816
C02480=1047.318,134.671,411.154,170.763,36.222,156.816
C02481=1047.311,134.422,411.176,170.761,36.220,156.815
C02482=1047.306,134.174,411.197,170.760,36.218,156.815
C02483=1047.299,133.924,411.218,170.758,36.216,156.814
C02484=1047.293,133.675,411.239,170.755,36.215,156.814
C02485=1047.288,133.426,411.261,170.753,36.213,156.814
C02486=1047.281,133.177,411.281,170.751,36.211,156.814
C02487=1047.275,132.928,411.303,170.750,36.209,156.813
C02488=1047.269,132.679,411.324,170.748,36.207,156.813
C02489=1047.263,132.430,411.344,170.746,36.206,156.813
C02490=1047.257,132.181,411.365,170.743,36.204,156.812
C02491=1047.251,131.931,411.386,170.742,36.202,156.812
C02492=1047.245,131.683,411.407,170.740,36.200,156.812
C02493=1047.239,131.434,411.429,170.738,36.199,156.811
C02494=1047.233,131.184,411.450,170.736,36.197,156.811
C02495=1047.227,130.936,411.470,170.734,36.195,156.811
C02496=1047.220,130.686,411.491,170.732,36.194,156.810
C02497=1047.214,130.437,411.512,170.730,36.192,156.810
C02498=1047.208,130.188,411.532,170.728,36.190,156.810
C02499=1047.201,129.939,411.553,170.726,36.189,156.809
C02500=1047.196,129.690,411.574,170.725,36.187,156.809
C02501=1047.189,129.441,411.595,170.722,36.185,156.809
C02502=1047.183,129.192,411.616,170.720,36.184,156.808
C02503=1047.177,128.943,411.636,170.718,36.182,156.808
C02504=1047.170,128.694,411.657,170.717,36.181,156.808
C02505=1047.165,128.445,411.677,170.715,36.179,156.807
C02506=1047.158,128.196,411.698,170.713,36.177,156.807
C02507=1047.152,127.947,411.718,170.710,36.176,156.807
C02508=1047.146,127.698,411.740,170.708,36.174,156.807
C02509=1047.139,127.448,411.760,170.707,36.172,156.806
C02510=1047.133,127.200,411.780,170.705,36.171,156.806
C02511=1047.127,126.950,411.802,170.703,36.169,156.806
C02512=1047.121,126.702,411.822,170.701,36.167,156.805
C02513=1047.115,126.452,411.843,170.699,36.166,156.805
C02514=1047.109,126.204,411.863,170.697,36.164,156.805
C02515=1047.101,125.917,411.887,170.695,36.162,156.804
C02516=1047.094,125.632,411.911,170.693,36.161,156.804
C02517=1047.087,125.346,411.934,170.691,36.159,156.804
C02518=1047.080,125.061,411.958,170.688,36.157,156.803
C02519=1047.075,124.811,411.979,170.686,36.155,156.803
C02520=1047.068,124.563,411.999,170.684,36.153,156.802
C02521=1047.062,124.313,412.020,170.683,36.151,156.802
C02522=1047.056,124.064,412.040,170.681,36.150,156.802
C02523=1047.050,123.815,412.061,170.679,36.148,156.802
C02524=1047.044,123.566,412.081,170.676,36.146,156.801
C02525=1047.038,123.316,412.102,170.675,36.145,156.801
C02526=1047.032,123.068,412.122,170.673,36.143,156.801
C02527=1047.025,122.819,412.143,170.671,36.141,156.800
C02528=1047.019,122.570,412.163,170.669,36.140,156.800
C02529=1047.013,122.320,412.184,170.668,36.138,156.800
C02530=1047.007,122.071,412.204,170.665,36.136,156.799
C02531=1047.000,121.822,412.225,170.663,36.135,156.799
C02532=1046.995,121.573,412.246,170.662,36.133,156.799
C02533=1046.988,121.324,412.266,170.660,36.131,156.798
C02534=1046.982,121.075,412.286,170.658,36.130,156.798
C02535=1046.977,120.826,412.306,170.656,36.128,156.798
C02536=1046.970,120.577,412.327,170.654,36.126,156.797
C02537=1046.964,120.328,412.347,170.652,36.125,156.797
C02538=1046.958,120.078,412.368,170.650,36.123,156.797
C02539=1046.952,119.829,412.388,170.649,36.121,156.796
C02540=1046.946,119.581,412.408,170.647,36.120,156.796
C02541=1046.940,119.331,412.429,170.645,36.118,156.796
C02542=1046.934,119.082,412.449,170.642,36.116,156.796
C02543=1046.927,118.833,412.470,170.641,36.114,156.795
C02544=1046.921,118.584,412.490,170.639,36.113,156.795
C02545=1046.916,118.335,412.511,170.637,36.111,156.795
C02546=1046.910,118.086,412.531,170.636,36.109,156.794
C02547=1046.904,117.837,412.551,170.634,36.108,156.794
C02548=1046.898,117.588,412.571,170.631,36.106,156.794
C02549=1046.892,117.338,412.592,170.629,36.104,156.793
C02550=1046.886,117.089,412.612,170.628,36.102,156.793
C02551=1046.880,116.841,412.632,170.626,36.101,156.793
C02552=1046.874,116.591,412.653,170.624,36.099,156.792
C02553=1046.868,116.342,412.673,170.622,36.097,156.792
C02554=1046.862,116.093,412.693,170.620,36.096,156.792
C02555=1046.856,115.844,412.714,170.618,36.094,156.791
C02556=1046.850,115.595,412.734,170.617,36.092,156.791
C02557=1046.844,115.346,412.754,170.615,36.091,156.791
C02558=1046.837,115.097,412.774,170.613,36.089,156.790
C02559=1046.832,114.848,412.795,170.611,36.087,156.790
C02560=1046.826,114.599,412.815,170.609,36.086,156.790
C02561=1046.819,114.349,412.835,170.607,36.084,156.790
C02562=1046.813,114.101,412.855,170.606,36.082,156.789
C02563=1046.808,113.851,412.875,170.604,36.081,156.789
C02564=1046.802,113.601,412.895,170.602,36.079,156.788
C02565=1046.796,113.352,412.915,170.599,36.077,156.788
C02566=1046.790,113.104,412.935,170.598,36.076,156.788
C02567=1046.783,112.854,412.956,170.596,36.074,156.788
C02568=1046.777,112.605,412.976,170.594,36.072,156.787
C02569=1046.771,112.356,412.996,170.593,36.071,156.787
C02570=1046.765,112.107,413.016,170.591,36.069,156.787
C02571=1046.759,111.858,413.036,170.588,36.067,156.786
C02572=1046.753,111.609,413.055,170.587,36.066,156.786
C02573=1046.747,111.360,413.075,170.585,36.064,156.786
C02574=1046.740,111.110,413.095,170.583,36.062,156.785
C02575=1046.734,110.862,413.115,170.582,36.061,156.785
C02576=1046.728,110.613,413.135,170.580,36.059,156.785
C02577=1046.722,110.363,413.156,170.578,36.058,156.785
C02578=1046.716,110.114,413.175,170.575,36.056,156.784
C02579=1046.709,109.828,413.197,170.573,36.054,156.784
C02580=1046.702,109.542,413.220,170.572,36.052,156.784
C02581=1046.695,109.256,413.242,170.570,36.050,156.783
C02582=1046.688,108.971,413.266,170.568,36.049,156.783
C02583=1046.681,108.721,413.286,170.566,36.047,156.783
C02584=1046.674,108.472,413.305,170.563,36.045,156.782
C02585=1046.668,108.224,413.325,170.562,36.044,156.782
C02586=1046.663,107.974,413.344,170.560,36.042,156.782
C02587=1046.656,107.725,413.365,170.558,36.041,156.781
C02588=1046.650,107.476,413.385,170.556,36.039,156.781
C02589=1046.644,107.227,413.405,170.555,36.038,156.781
C02590=1046.638,106.977,413.424,170.552,36.036,156.780
C02591=1046.631,106.728,413.444,170.550,36.035,156.780
C02592=1046.625,106.480,413.463,170.549,36.033,156.780
C02593=1046.620,106.230,413.483,170.547,36.031,156.780
C02594=1046.614,105.981,413.503,170.545,36.030,156.779
C02595=1046.607,105.731,413.522,170.544,36.028,156.779
C02596=1046.601,105.482,413.542,170.542,36.027,156.779
C02597=1046.595,105.234,413.562,170.539,36.025,156.778
C02598=1046.589,104.984,413.581,170.538,36.023,156.778
C02599=1046.582,104.735,413.601,170.536,36.022,156.778
C02600=1046.576,104.486,413.621,170.534,36.020,156.778
C02601=1046.571,104.237,413.640,170.533,36.018,156.777
C02602=1046.565,103.988,413.660,170.531,36.017,156.777
C02603=1046.558,103.739,413.679,170.528,36.015,156.777
C02604=1046.552,103.489,413.699,170.527,36.013,156.776
C02605=1046.546,103.240,413.719,170.525,36.012,156.776
C02606=1046.540,102.991,413.739,170.523,36.010,156.776
C02607=1046.534,102.742,413.758,170.522,36.009,156.775
C02608=1046.528,102.493,413.778,170.520,36.007,156.775
C02609=1046.521,102.244,413.797,170.517,36.005,156.775
C02610=1046.515,101.994,413.817,170.516,36.004,156.774
C02611=1046.509,101.745,413.837,170.514,36.002,156.774
C02612=1046.503,101.496,413.856,170.512,36.001,156.774
C02613=1046.497,101.247,413.876,170.511,35.999,156.774
C02614=1046.491,100.998,413.894,170.509,35.997,156.773
C02615=1046.485,100.749,413.914,170.507,35.996,156.773
C02616=1046.479,100.500,413.934,170.505,35.994,156.773
C02617=1046.473,100.250,413.954,170.503,35.993,156.772
C02618=1046.466,100.001,413.973,170.501,35.991,156.772
C02619=1046.461,99.752,413.992,170.500,35.990,156.772
C02620=1046.454,99.503,414.011,170.498,35.988,156.771
C02621=1046.448,99.254,414.031,170.496,35.986,156.771
C02622=1046.441,99.004,414.050,170.494,35.984,156.771
C02623=1046.435,98.755,414.069,170.492,35.983,156.771
C02624=1046.429,98.506,414.088,170.490,35.982,156.770
C02625=1046.423,98.257,414.108,170.489,35.980,156.770
C02626=1046.417,98.008,414.127,170.487,35.979,156.770
C02627=1046.411,97.759,414.146,170.485,35.977,156.769
C02628=1046.405,97.510,414.166,170.484,35.976,156.769
C02629=1046.398,97.260,414.185,170.481,35.974,156.769
C02630=1046.392,97.010,414.204,170.479,35.972,156.769
C02631=1046.385,96.762,414.224,170.478,35.971,156.768
C02632=1046.380,96.512,414.243,170.476,35.969,156.768
C02633=1046.373,96.263,414.261,170.474,35.967,156.768
C02634=1046.367,96.015,414.281,170.473,35.966,156.767
C02635=1046.361,95.765,414.301,170.471,35.964,156.767
C02636=1046.355,95.516,414.319,170.468,35.963,156.767
C02637=1046.349,95.267,414.339,170.467,35.961,156.767
C02638=1046.342,95.017,414.358,170.465,35.960,156.766
C02639=1046.336,94.768,414.378,170.463,35.958,156.766
C02640=1046.330,94.519,414.396,170.462,35.957,156.766
C02641=1046.324,94.269,414.415,170.460,35.955,156.765
C02642=1046.317,94.021,414.435,170.458,35.954,156.765
C02643=1046.310,93.735,414.456,170.455,35.952,156.765
C02644=1046.304,93.449,414.479,170.454,35.950,156.764
C02645=1046.297,93.163,414.501,170.452,35.948,156.764
C02646=1046.290,92.877,414.523,170.450,35.946,156.764
C02647=1046.283,92.628,414.542,170.448,35.945,156.764
C02648=1046.278,92.379,414.561,170.446,35.943,156.763
C02649=1046.271,92.130,414.580,170.444,35.942,156.763
C02650=1046.265,91.880,414.599,170.442,35.940,156.763
C02651=1046.259,91.631,414.617,170.441,35.938,156.762
C02652=1046.253,91.382,414.637,170.439,35.937,156.762
C02653=1046.247,91.133,414.656,170.437,35.935,156.762
C02654=1046.241,90.884,414.675,170.436,35.933,156.761
C02655=1046.234,90.634,414.694,170.434,35.931,156.761
C02656=1046.229,90.385,414.713,170.431,35.930,156.761
C02657=1046.222,90.136,414.732,170.430,35.929,156.761
C02658=1046.217,89.887,414.751,170.428,35.927,156.760
C02659=1046.210,89.637,414.770,170.426,35.926,156.760
C02660=1046.204,89.388,414.788,170.425,35.924,156.760
C02661=1046.197,89.139,414.807,170.423,35.923,156.759
C02662=1046.192,88.890,414.826,170.421,35.921,156.759
C02663=1046.185,88.641,414.845,170.419,35.919,156.759
C02664=1046.179,88.391,414.864,170.417,35.918,156.759
C02665=1046.172,88.142,414.882,170.415,35.916,156.758
C02666=1046.166,87.892,414.902,170.414,35.915,156.758
C02667=1046.160,87.643,414.920,170.412,35.914,156.758
C02668=1046.153,87.394,414.939,170.410,35.912,156.758
C02669=1046.147,87.145,414.958,170.409,35.911,156.757
C02670=1046.141,86.895,414.977,170.406,35.909,156.757
C02671=1046.135,86.646,414.996,170.404,35.907,156.757
C02672=1046.128,86.397,415.014,170.403,35.906,156.756
C02673=1046.122,86.148,415.033,170.401,35.904,156.756
C02674=1046.116,85.900,415.051,170.399,35.903,156.756
C02675=1046.110,85.650,415.070,170.398,35.901,156.756
C02676=1046.104,85.401,415.089,170.396,35.900,156.755
C02677=1046.098,85.152,415.108,170.393,35.898,156.755
C02678=1046.091,84.903,415.126,170.392,35.897,156.755
C02679=1046.085,84.653,415.146,170.390,35.895,156.755
C02680=1046.079,84.404,415.164,170.389,35.893,156.754
C02681=1046.073,84.155,415.183,170.387,35.892,156.754
C02682=1046.066,83.905,415.201,170.385,35.890,156.754
C02683=1046.061,83.656,415.220,170.384,35.889,156.753
C02684=1046.054,83.407,415.239,170.382,35.888,156.753
C02685=1046.048,83.158,415.257,170.379,35.886,156.753
C02686=1046.041,82.909,415.276,170.378,35.885,156.753
C02687=1046.035,82.659,415.295,170.376,35.883,156.752
C02688=1046.029,82.410,415.314,170.374,35.881,156.752
C02689=1046.023,82.160,415.332,170.373,35.880,156.752
C02690=1046.017,81.911,415.351,170.371,35.878,156.751
C02691=1046.011,81.663,415.369,170.368,35.876,156.751
C02692=1046.005,81.414,415.387,170.367,35.875,156.751
C02693=1045.999,81.164,415.407,170.365,35.874,156.751
C02694=1045.993,80.914,415.425,170.363,35.872,156.750
C02695=1045.986,80.665,415.443,170.362,35.871,156.750
C02696=1045.980,80.416,415.462,170.360,35.869,156.750
C02697=1045.973,80.167,415.481,170.359,35.867,156.749
C02698=1045.968,79.917,415.499,170.357,35.866,156.749
C02699=1045.962,79.669,415.517,170.354,35.864,156.749
C02700=1045.956,79.420,415.536,170.353,35.862,156.748
C02701=1045.949,79.170,415.555,170.351,35.861,156.748
C02702=1045.943,78.921,415.573,170.349,35.859,156.748
C02703=1045.938,78.671,415.592,170.348,35.858,156.748
C02704=1045.931,78.422,415.611,170.346,35.857,156.747
C02705=1045.925,78.173,415.629,170.344,35.855,156.747
C02706=1045.919,77.924,415.647,170.342,35.854,156.747
C02707=1045.911,77.638,415.668,170.340,35.852,156.747
C02708=1045.904,77.352,415.689,170.338,35.850,156.746
C02709=1045.897,77.066,415.710,170.336,35.848,156.746
C02710=1045.890,76.780,415.732,170.334,35.847,156.746
C02711=1045.884,76.531,415.749,170.333,35.845,156.745
C02712=1045.878,76.282,415.768,170.331,35.843,156.745
C02713=1045.872,76.032,415.786,170.328,35.842,156.745
C02714=1045.865,75.783,415.804,170.327,35.840,156.744
C02715=1045.859,75.534,415.823,170.325,35.839,156.744
C02716=1045.853,75.284,415.841,170.323,35.838,156.744
C02717=1045.846,75.035,415.859,170.322,35.836,156.744
C02718=1045.840,74.786,415.877,170.320,35.834,156.743
C02719=1045.834,74.537,415.895,170.318,35.833,156.743
C02720=1045.828,74.287,415.913,170.316,35.831,156.743
C02721=1045.821,74.038,415.932,170.314,35.830,156.743
C02722=1045.815,73.788,415.950,170.312,35.829,156.742
C02723=1045.809,73.540,415.968,170.311,35.827,156.742
C02724=1045.803,73.290,415.986,170.309,35.826,156.742
C02725=1045.797,73.041,416.005,170.307,35.824,156.741
C02726=1045.790,72.792,416.023,170.306,35.822,156.741
C02727=1045.784,72.542,416.041,170.304,35.821,156.741
C02728=1045.779,72.293,416.059,170.302,35.819,156.741
C02729=1045.772,72.044,416.077,170.300,35.818,156.740
C02730=1045.766,71.794,416.095,170.298,35.817,156.740
C02731=1045.759,71.546,416.113,170.297,35.815,156.740
C02732=1045.753,71.296,416.131,170.295,35.813,156.740
C02733=1045.747,71.047,416.150,170.293,35.812,156.739
C02734=1045.741,70.798,416.168,170.292,35.810,156.739
C02735=1045.734,70.549,416.186,170.290,35.809,156.739
C02736=1045.728,70.299,416.204,170.287,35.807,156.739
C02737=1045.722,70.050,416.222,170.286,35.806,156.738
C02738=1045.716,69.801,416.240,170.284,35.805,156.738
C02739=1045.709,69.551,416.258,170.282,35.803,156.738
C02740=1045.703,69.302,416.276,170.281,35.801,156.737
C02741=1045.698,69.053,416.294,170.279,35.800,156.737
C02742=1045.691,68.803,416.312,170.277,35.798,156.737
C02743=1045.685,68.554,416.331,170.275,35.797,156.737
C02744=1045.678,68.305,416.348,170.273,35.796,156.736
C02745=1045.673,68.056,416.365,170.272,35.794,156.736
C02746=1045.666,67.807,416.384,170.270,35.792,156.736
C02747=1045.660,67.557,416.402,170.268,35.791,156.736
C02748=1045.653,67.307,416.419,170.267,35.789,156.735
C02749=1045.647,67.059,416.438,170.265,35.788,156.735
C02750=1045.641,66.809,416.456,170.263,35.787,156.735
C02751=1045.634,66.560,416.473,170.261,35.785,156.734
C02752=1045.629,66.311,416.491,170.259,35.783,156.734
C02753=1045.622,66.062,416.509,170.257,35.782,156.734
C02754=1045.616,65.812,416.527,170.256,35.781,156.734
C02755=1045.609,65.563,416.544,170.254,35.779,156.733
C02756=1045.604,65.314,416.563,170.252,35.778,156.733
C02757=1045.598,65.064,416.581,170.251,35.776,156.733
C02758=1045.591,64.815,416.598,170.249,35.775,156.733
C02759=1045.585,64.566,416.616,170.246,35.773,156.732
C02760=1045.579,64.316,416.633,170.245,35.772,156.732
C02761=1045.572,64.067,416.652,170.243,35.770,156.732
C02762=1045.566,63.818,416.669,170.241,35.769,156.732
C02763=1045.559,63.569,416.686,170.240,35.768,156.731
C02764=1045.553,63.319,416.704,170.238,35.766,156.731
C02765=1045.547,63.070,416.722,170.236,35.765,156.731
C02766=1045.541,62.821,416.739,170.235,35.763,156.731
C02767=1045.534,62.571,416.757,170.232,35.762,156.730
C02768=1045.528,62.322,416.775,170.230,35.760,156.730
C02769=1045.521,62.073,416.793,170.229,35.759,156.730
C02770=1045.515,61.824,416.810,170.227,35.758,156.730
C02771=1045.507,61.537,416.830,170.225,35.756,156.729
C02772=1045.500,61.251,416.850,170.223,35.755,156.729
C02773=1045.492,60.965,416.870,170.221,35.753,156.729
C02774=1045.486,60.679,416.890,170.219,35.751,156.729
C02775=1045.479,60.429,416.908,170.217,35.750,156.728
C02776=1045.473,60.180,416.925,170.215,35.748,156.728
C02777=1045.466,59.931,416.942,170.213,35.747,156.728
C02778=1045.460,59.681,416.960,170.211,35.746,156.728
C02779=1045.454,59.432,416.977,170.210,35.744,156.727
C02780=1045.448,59.183,416.995,170.208,35.743,156.727
C02781=1045.441,58.933,417.013,170.206,35.741,156.727
C02782=1045.435,58.685,417.030,170.205,35.740,156.727
C02783=1045.429,58.435,417.047,170.203,35.739,156.726
C02784=1045.422,58.185,417.065,170.200,35.737,156.726
C02785=1045.416,57.936,417.082,170.199,35.735,156.726
C02786=1045.409,57.687,417.100,170.197,35.734,156.726
C02787=1045.402,57.437,417.117,170.195,35.733,156.725
C02788=1045.397,57.188,417.135,170.194,35.732,156.725
C02789=1045.390,56.939,417.152,170.192,35.730,156.725
C02790=1045.385,56.690,417.169,170.190,35.728,156.724
C02791=1045.378,56.441,417.187,170.189,35.727,156.724
C02792=1045.371,56.191,417.204,170.187,35.726,156.724
C02793=1045.365,55.942,417.222,170.184,35.725,156.724
C02794=1045.358,55.693,417.239,170.183,35.723,156.724
C02795=1045.353,55.444,417.257,170.181,35.721,156.723
C02796=1045.346,55.194,417.274,170.179,35.720,156.723
C02797=1045.340,54.945,417.290,170.178,35.719,156.723
C02798=1045.334,54.695,417.308,170.176,35.718,156.723
C02799=1045.327,54.446,417.326,170.174,35.716,156.722
C02800=1045.322,54.197,417.343,170.173,35.714,156.722
C02801=1045.315,53.947,417.360,170.170,35.713,156.722
C02802=1045.309,53.698,417.377,170.168,35.712,156.722
C02803=1045.302,53.449,417.395,170.167,35.710,156.721
C02804=1045.296,53.200,417.412,170.165,35.709,156.721
C02805=1045.290,52.950,417.429,170.163,35.707,156.721
C02806=1045.284,52.701,417.446,170.162,35.706,156.721
C02807=1045.277,52.451,417.464,170.160,35.704,156.720
C02808=1045.272,52.202,417.481,170.158,35.703,156.720
C02809=1045.265,51.953,417.499,170.156,35.701,156.720
C02810=1045.259,51.704,417.515,170.154,35.700,156.719
C02811=1045.253,51.454,417.533,170.152,35.699,156.719
C02812=1045.247,51.205,417.550,170.151,35.697,156.719
C02813=1045.240,50.956,417.567,170.149,35.696,156.719
C02814=1045.234,50.707,417.585,170.147,35.694,156.718
C02815=1045.228,50.457,417.601,170.146,35.693,156.718
C02816=1045.221,50.208,417.618,170.144,35.691,156.718
C02817=1045.215,49.958,417.636,170.142,35.690,156.718
C02818=1045.209,49.709,417.653,170.140,35.689,156.717
C02819=1045.202,49.459,417.670,170.138,35.687,156.717
C02820=1045.197,49.210,417.687,170.136,35.685,156.717
C02821=1045.190,48.961,417.705,170.135,35.684,156.717
C02822=1045.184,48.712,417.721,170.133,35.683,156.716
C02823=1045.178,48.462,417.739,170.131,35.681,156.716
C02824=1045.172,48.213,417.756,170.130,35.680,156.716
C02825=1045.165,47.963,417.773,170.128,35.678,156.716
C02826=1045.160,47.714,417.790,170.126,35.677,156.715
C02827=1045.153,47.465,417.807,170.123,35.675,156.715
C02828=1045.147,47.215,417.824,170.122,35.674,156.715
C02829=1045.141,46.966,417.841,170.120,35.673,156.715
C02830=1045.134,46.717,417.859,170.118,35.671,156.714
C02831=1045.128,46.467,417.875,170.117,35.669,156.714
C02832=1045.123,46.218,417.892,170.115,35.668,156.714
C02833=1045.116,45.969,417.910,170.113,35.667,156.714
C02834=1045.110,45.720,417.926,170.112,35.665,156.713
C02835=1045.103,45.446,417.945,170.109,35.664,156.713
C02836=1045.097,45.173,417.964,170.107,35.662,156.713
C02837=1045.090,44.900,417.982,170.105,35.660,156.712
C02838=1045.084,44.627,418.001,170.103,35.658,156.712
C02839=1045.077,44.377,418.018,170.102,35.657,156.712
C02840=1045.071,44.129,418.035,170.100,35.656,156.712
C02841=1045.065,43.879,418.052,170.098,35.655,156.711
C02842=1045.059,43.630,418.069,170.097,35.653,156.711
C02843=1045.053,43.380,418.086,170.094,35.651,156.711
C02844=1045.046,43.132,418.103,170.092,35.650,156.711
C02845=1045.040,42.882,418.119,170.091,35.649,156.710
C02846=1045.034,42.633,418.137,170.089,35.647,156.710
C02847=1045.028,42.382,418.153,170.087,35.646,156.710
C02848=1045.021,42.134,418.170,170.086,35.644,156.710
C02849=1045.016,41.884,418.187,170.084,35.643,156.709
C02850=1045.009,41.635,418.204,170.082,35.642,156.709
C02851=1045.003,41.386,418.220,170.081,35.640,156.709
C02852=1044.996,41.136,418.237,170.078,35.639,156.709
C02853=1044.990,40.887,418.254,170.076,35.637,156.708
C02854=1044.984,40.637,418.270,170.074,35.636,156.708
C02855=1044.977,40.374,418.288,170.073,35.635,156.708
C02856=1044.970,40.112,418.306,170.071,35.633,156.708
C02857=1044.964,39.849,418.324,170.069,35.631,156.707
C02858=1044.957,39.586,418.341,170.067,35.630,156.707
C02859=1044.951,39.338,418.357,170.066,35.629,156.707
C02860=1044.944,39.088,418.374,170.064,35.627,156.707
C02861=1044.938,38.838,418.390,170.061,35.626,156.707
C02862=1044.933,38.589,418.408,170.059,35.624,156.706
C02863=1044.926,38.339,418.425,170.058,35.623,156.706
C02864=1044.920,38.090,418.441,170.056,35.622,156.706
C02865=1044.914,37.841,418.458,170.054,35.620,156.706
C02866=1044.908,37.591,418.474,170.053,35.619,156.705
C02867=1044.902,37.342,418.491,170.051,35.618,156.705
C02868=1044.895,37.093,418.507,170.049,35.616,156.705
C02869=1044.888,36.843,418.524,170.048,35.615,156.705
C02870=1044.882,36.594,418.540,170.045,35.613,156.704
C02871=1044.876,36.344,418.556,170.043,35.612,156.704
C02872=1044.869,36.095,418.574,170.041,35.611,156.704
C02873=1044.863,35.846,418.590,170.040,35.609,156.704
C02874=1044.857,35.597,418.605,170.038,35.608,156.703
C02875=1044.850,35.347,418.622,170.036,35.607,156.703
C02876=1044.844,35.098,418.639,170.034,35.605,156.703
C02877=1044.838,34.849,418.655,170.033,35.604,156.703
C02878=1044.832,34.599,418.672,170.031,35.603,156.703
C02879=1044.825,34.349,418.688,170.029,35.602,156.702
C02880=1044.819,34.100,418.704,170.027,35.600,156.702
C02881=1044.813,33.851,418.721,170.025,35.599,156.702
C02882=1044.806,33.601,418.737,170.023,35.598,156.702
C02883=1044.800,33.352,418.754,170.021,35.596,156.701
C02884=1044.794,33.103,418.770,170.020,35.594,156.701
C02885=1044.788,32.853,418.786,170.018,35.593,156.701
C02886=1044.781,32.604,418.802,170.016,35.592,156.701
C02887=1044.775,32.355,418.819,170.014,35.591,156.700
C02888=1044.769,32.105,418.835,170.013,35.589,156.700
C02889=1044.763,31.856,418.852,170.011,35.588,156.700
C02890=1044.756,31.606,418.868,170.008,35.587,156.700
C02891=1044.749,31.357,418.884,170.007,35.585,156.699
C02892=1044.743,31.108,418.900,170.005,35.584,156.699
C02893=1044.738,30.858,418.917,170.003,35.583,156.699
C02894=1044.731,30.608,418.933,170.001,35.581,156.699
C02895=1044.725,30.359,418.949,170.000,35.579,156.698
C02896=1044.718,30.110,418.966,169.998,35.578,156.698
C02897=1044.712,29.861,418.982,169.996,35.577,156.698
C02898=1044.706,29.612,418.998,169.994,35.576,156.698
C02899=1044.699,29.325,419.016,169.992,35.574,156.698
C02900=1044.692,29.038,419.036,169.989,35.572,156.697
C02901=1044.684,28.751,419.054,169.987,35.571,156.697
C02902=1044.677,28.465,419.073,169.985,35.570,156.697
C02903=1044.671,28.216,419.089,169.984,35.568,156.697
C02904=1044.664,27.967,419.105,169.982,35.567,156.696
C02905=1044.658,27.717,419.121,169.980,35.566,156.696
C02906=1044.652,27.467,419.137,169.978,35.565,156.696
C02907=1044.645,27.218,419.153,169.977,35.563,156.696
C02908=1044.640,26.968,419.169,169.975,35.562,156.695
C02909=1044.633,26.719,419.185,169.972,35.561,156.695
C02910=1044.627,26.470,419.201,169.970,35.559,156.695
C02911=1044.621,26.221,419.217,169.969,35.558,156.695
C02912=1044.614,25.971,419.233,169.967,35.557,156.695
C02913=1044.608,25.722,419.250,169.965,35.555,156.694
C02914=1044.601,25.473,419.265,169.963,35.554,156.694
C02915=1044.595,25.223,419.281,169.962,35.553,156.694
C02916=1044.589,24.974,419.298,169.960,35.551,156.694
C02917=1044.582,24.724,419.314,169.958,35.550,156.694
C02918=1044.576,24.474,419.329,169.956,35.549,156.693
C02919=1044.569,24.225,419.345,169.955,35.548,156.693
C02920=1044.564,23.976,419.361,169.952,35.546,156.693
C02921=1044.557,23.727,419.377,169.950,35.545,156.693
C02922=1044.551,23.477,419.393,169.948,35.544,156.692
C02923=1044.545,23.228,419.409,169.947,35.542,156.692
C02924=1044.538,22.978,419.425,169.945,35.541,156.692
C02925=1044.532,22.728,419.441,169.943,35.540,156.692
C02926=1044.525,22.479,419.457,169.941,35.538,156.692
C02927=1044.519,22.230,419.473,169.939,35.537,156.691
C02928=1044.513,21.981,419.489,169.938,35.536,156.691
C02929=1044.507,21.731,419.504,169.936,35.535,156.691
C02930=1044.500,21.482,419.520,169.933,35.533,156.691
C02931=1044.494,21.233,419.536,169.931,35.532,156.690
C02932=1044.488,20.983,419.552,169.930,35.531,156.690
C02933=1044.482,20.734,419.567,169.928,35.529,156.690
C02934=1044.475,20.483,419.584,169.926,35.528,156.690
C02935=1044.469,20.234,419.599,169.924,35.527,156.690
C02936=1044.463,19.985,419.616,169.923,35.525,156.689
C02937=1044.456,19.735,419.631,169.921,35.524,156.689
C02938=1044.451,19.486,419.647,169.919,35.523,156.689
C02939=1044.444,19.237,419.663,169.917,35.521,156.689
C02940=1044.437,18.987,419.678,169.915,35.520,156.688
C02941=1044.431,18.738,419.694,169.913,35.519,156.688
C02942=1044.425,18.489,419.709,169.911,35.518,156.688
C02943=1044.419,18.239,419.725,169.909,35.516,156.688
C02944=1044.412,17.990,419.741,169.907,35.515,156.688
C02945=1044.406,17.741,419.756,169.905,35.514,156.687
C02946=1044.400,17.490,419.772,169.904,35.512,156.687
C02947=1044.393,17.241,419.788,169.902,35.511,156.687
C02948=1044.387,16.992,419.804,169.900,35.510,156.687
C02949=1044.381,16.742,419.819,169.898,35.509,156.687
C02950=1044.374,16.493,419.835,169.897,35.508,156.686
C02951=1044.368,16.243,419.850,169.895,35.506,156.686
C02952=1044.361,15.994,419.866,169.892,35.505,156.686
C02953=1044.356,15.745,419.882,169.890,35.504,156.686
C02954=1044.349,15.495,419.897,169.888,35.502,156.685
C02955=1044.342,15.246,419.913,169.887,35.501,156.685
C02956=1044.337,14.996,419.928,169.885,35.500,156.685
C02957=1044.330,14.747,419.944,169.883,35.499,156.685
C02958=1044.324,14.497,419.960,169.881,35.497,156.685
C02959=1044.318,14.248,419.975,169.879,35.496,156.684
C02960=1044.311,13.998,419.990,169.878,35.495,156.684
C02961=1044.305,13.749,420.006,169.876,35.494,156.684
C02962=1044.298,13.500,420.021,169.874,35.493,156.684
C02963=1044.292,13.214,420.039,169.871,35.491,156.684
C02964=1044.284,12.929,420.057,169.869,35.490,156.683
C02965=1044.276,12.644,420.074,169.867,35.489,156.683
C02966=1044.270,12.359,420.092,169.865,35.487,156.683
C02967=1044.263,12.110,420.107,169.863,35.486,156.683
C02968=1044.257,11.860,420.122,169.861,35.485,156.683
C02969=1044.250,11.611,420.137,169.859,35.483,156.682
C02970=1044.244,11.361,420.152,169.857,35.482,156.682
C02971=1044.238,11.112,420.168,169.855,35.481,156.682
C02972=1044.231,10.862,420.183,169.854,35.480,156.682
C02973=1044.225,10.613,420.198,169.852,35.479,156.682
C02974=1044.218,10.364,420.214,169.850,35.477,156.681
C02975=1044.212,10.114,420.229,169.847,35.476,156.681
C02976=1044.205,9.865,420.245,169.845,35.475,156.681
C02977=1044.199,9.615,420.260,169.843,35.474,156.681
C02978=1044.192,9.366,420.275,169.842,35.473,156.681
C02979=1044.186,9.116,420.291,169.840,35.472,156.680
C02980=1044.180,8.867,420.306,169.838,35.470,156.680
C02981=1044.174,8.617,420.321,169.836,35.469,156.680
C02982=1044.167,8.368,420.336,169.834,35.468,156.680
C02983=1044.161,8.118,420.351,169.832,35.467,156.680
C02984=1044.154,7.869,420.366,169.831,35.466,156.679
C02985=1044.148,7.619,420.381,169.829,35.464,156.679
C02986=1044.141,7.370,420.397,169.827,35.463,156.679
C02987=1044.135,7.120,420.412,169.824,35.462,156.679
C02988=1044.129,6.870,420.427,169.822,35.461,156.679
C02989=1044.123,6.621,420.442,169.820,35.460,156.678
C02990=1044.117,6.372,420.458,169.818,35.458,156.678
C02991=1044.110,6.123,420.473,169.817,35.457,156.678
C02992=1044.104,5.873,420.487,169.815,35.456,156.678
C02993=1044.098,5.623,420.502,169.813,35.455,156.678
C02994=1044.091,5.374,420.518,169.811,35.454,156.677
C02995=1044.084,5.125,420.533,169.809,35.452,156.677
C02996=1044.078,4.875,420.548,169.807,35.451,156.677
C02997=1044.072,4.626,420.563,169.806,35.450,156.677
C02998=1044.067,4.376,420.578,169.804,35.449,156.677
C02999=1044.060,4.127,420.594,169.801,35.448,156.676
C03000=1044.054,3.877,420.609,169.799,35.446,156.676
C03001=1044.047,3.628,420.624,169.797,35.445,156.676
C03002=1044.041,3.378,420.639,169.795,35.444,156.676
C03003=1044.034,3.128,420.654,169.793,35.443,156.676
C03004=1044.029,2.879,420.668,169.792,35.442,156.675
C03005=1044.022,2.630,420.684,169.790,35.441,156.675
C03006=1044.016,2.381,420.699,169.788,35.439,156.675
C03007=1044.009,2.131,420.714,169.786,35.438,156.675
C03008=1044.003,1.881,420.729,169.784,35.437,156.675
C03009=1043.997,1.632,420.743,169.782,35.436,156.674
C03010=1043.991,1.383,420.758,169.780,35.435,156.674
C03011=1043.984,1.133,420.773,169.779,35.433,156.674
C03012=1043.979,0.883,420.789,169.776,35.432,156.674
C03013=1043.972,0.633,420.804,169.774,35.431,156.674
C03014=1043.966,0.385,420.818,169.772,35.430,156.673
C03015=1043.960,0.135,420.833,169.770,35.429,156.673
C03016=1043.953,-0.114,420.849,169.768,35.427,156.673
C03017=1043.947,-0.364,420.864,169.766,35.426,156.673
C03018=1043.941,-0.613,420.878,169.765,35.425,156.673
C03019=1043.935,-0.862,420.893,169.763,35.424,156.673
C03020=1043.928,-1.112,420.908,169.761,35.423,156.672
C03021=1043.922,-1.362,420.923,169.759,35.421,156.672
C03022=1043.916,-1.611,420.938,169.757,35.420,156.672
C03023=1043.910,-1.860,420.953,169.755,35.419,156.672
C03024=1043.904,-2.110,420.968,169.752,35.418,156.672
C03025=1043.897,-2.360,420.983,169.750,35.417,156.671
C03026=1043.891,-2.609,420.997,169.749,35.415,156.671
C03027=1043.884,-2.892,421.013,169.746,35.414,156.671
C03028=1043.878,-3.176,421.030,169.744,35.413,156.671
C03029=1043.871,-3.459,421.047,169.742,35.411,156.670
C03030=1043.863,-3.742,421.064,169.740,35.410,156.670
C03031=1043.857,-3.992,421.079,169.738,35.409,156.670
C03032=1043.851,-4.242,421.094,169.736,35.408,156.670
C03033=1043.844,-4.491,421.108,169.734,35.407,156.670
C03034=1043.837,-4.741,421.123,169.732,35.405,156.670
C03035=1043.832,-4.990,421.137,169.731,35.405,156.669
C03036=1043.825,-5.239,421.151,169.729,35.403,156.669
C03037=1043.818,-5.489,421.166,169.726,35.403,156.669
C03038=1043.812,-5.739,421.181,169.724,35.401,156.669
C03039=1043.806,-5.988,421.196,169.722,35.400,156.669
C03040=1043.799,-6.237,421.210,169.720,35.399,156.669
C03041=1043.793,-6.487,421.224,169.718,35.398,156.668
C03042=1043.787,-6.736,421.239,169.716,35.397,156.668
C03043=1043.781,-6.986,421.254,169.714,35.396,156.668
C03044=1043.774,-7.235,421.268,169.712,35.395,156.668
C03045=1043.768,-7.486,421.282,169.710,35.394,156.668
C03046=1043.762,-7.735,421.297,169.708,35.393,156.667
C03047=1043.755,-7.984,421.311,169.706,35.391,156.667
C03048=1043.748,-8.234,421.326,169.705,35.391,156.667
C03049=1043.743,-8.483,421.340,169.703,35.389,156.667
C03050=1043.736,-8.732,421.355,169.701,35.389,156.667
C03051=1043.729,-8.982,421.369,169.699,35.387,156.667
C03052=1043.723,-9.231,421.384,169.696,35.386,156.666
C03053=1043.717,-9.481,421.398,169.694,35.385,156.666
C03054=1043.710,-9.731,421.413,169.692,35.384,156.666
C03055=1043.704,-9.980,421.427,169.690,35.383,156.666
C03056=1043.698,-10.230,421.441,169.688,35.382,156.666
C03057=1043.691,-10.479,421.456,169.686,35.381,156.666
C03058=1043.685,-10.728,421.470,169.684,35.380,156.665
C03059=1043.679,-10.978,421.485,169.682,35.379,156.665
C03060=1043.673,-11.227,421.499,169.680,35.377,156.665
C03061=1043.667,-11.477,421.514,169.678,35.377,156.665
C03062=1043.660,-11.727,421.528,169.676,35.375,156.665
C03063=1043.654,-11.976,421.542,169.675,35.375,156.665
C03064=1043.648,-12.225,421.557,169.673,35.373,156.664
C03065=1043.642,-12.475,421.571,169.671,35.372,156.664
C03066=1043.635,-12.724,421.585,169.669,35.371,156.664
C03067=1043.629,-12.975,421.599,169.666,35.370,156.664
C03068=1043.623,-13.224,421.614,169.664,35.369,156.664
C03069=1043.616,-13.473,421.628,169.662,35.368,156.664
C03070=1043.610,-13.722,421.642,169.660,35.367,156.663
C03071=1043.604,-13.972,421.657,169.658,35.366,156.663
C03072=1043.598,-14.221,421.670,169.656,35.365,156.663
C03073=1043.591,-14.471,421.685,169.654,35.363,156.663
C03074=1043.585,-14.721,421.699,169.652,35.363,156.663
C03075=1043.579,-14.970,421.713,169.650,35.361,156.663
C03076=1043.573,-15.220,421.728,169.648,35.360,156.662
C03077=1043.567,-15.469,421.742,169.646,35.359,156.662
C03078=1043.560,-15.719,421.756,169.644,35.358,156.662
C03079=1043.554,-15.968,421.770,169.642,35.357,156.662
C03080=1043.548,-16.218,421.784,169.640,35.356,156.662
C03081=1043.541,-16.467,421.798,169.638,35.355,156.662
C03082=1043.535,-16.717,421.812,169.635,35.354,156.661
C03083=1043.528,-16.966,421.827,169.633,35.353,156.661
C03084=1043.522,-17.216,421.840,169.631,35.352,156.661
C03085=1043.516,-17.466,421.854,169.629,35.351,156.661
C03086=1043.509,-17.715,421.868,169.627,35.350,156.661
C03087=1043.503,-17.965,421.882,169.625,35.349,156.661
C03088=1043.496,-18.213,421.896,169.623,35.348,156.661
C03089=1043.490,-18.464,421.910,169.621,35.348,156.660
C03090=1043.484,-18.714,421.924,169.619,35.346,156.660
C03091=1043.477,-18.995,421.940,169.617,35.345,156.660
C03092=1043.469,-19.277,421.956,169.615,35.344,156.660
C03093=1043.463,-19.558,421.971,169.613,35.343,156.660
C03094=1043.455,-19.840,421.987,169.610,35.342,156.660
C03095=1043.450,-20.090,422.001,169.608,35.341,156.659
C03096=1043.442,-20.339,422.015,169.606,35.340,156.659
C03097=1043.436,-20.588,422.029,169.604,35.339,156.659
C03098=1043.430,-20.839,422.043,169.602,35.338,156.659
C03099=1043.424,-21.087,422.057,169.599,35.337,156.659
C03100=1043.418,-21.338,422.071,169.597,35.336,156.659
C03101=1043.411,-21.587,422.084,169.595,35.335,156.658
C03102=1043.405,-21.837,422.098,169.593,35.334,156.658
C03103=1043.399,-22.086,422.112,169.591,35.333,156.658
C03104=1043.392,-22.336,422.126,169.589,35.332,156.658
C03105=1043.386,-22.585,422.140,169.587,35.331,156.658
C03106=1043.380,-22.835,422.154,169.585,35.330,156.658
C03107=1043.373,-23.084,422.168,169.583,35.329,156.658
C03108=1043.368,-23.333,422.181,169.581,35.328,156.657
C03109=1043.361,-23.583,422.195,169.579,35.327,156.657
C03110=1043.355,-23.833,422.208,169.577,35.326,156.657
C03111=1043.348,-24.082,422.223,169.575,35.325,156.657
C03112=1043.342,-24.332,422.237,169.573,35.324,156.657
C03113=1043.337,-24.581,422.250,169.571,35.323,156.657
C03114=1043.330,-24.831,422.264,169.569,35.323,156.657
C03115=1043.323,-25.080,422.277,169.567,35.321,156.656
C03116=1043.317,-25.331,422.292,169.564,35.320,156.656
C03117=1043.311,-25.579,422.306,169.562,35.319,156.656
C03118=1043.305,-25.829,422.319,169.560,35.318,156.656
C03119=1043.299,-26.079,422.333,169.558,35.317,156.656
C03120=1043.292,-26.328,422.346,169.556,35.316,156.656
C03121=1043.286,-26.577,422.360,169.554,35.316,156.656
C03122=1043.280,-26.828,422.374,169.552,35.314,156.655
C03123=1043.274,-27.077,422.387,169.550,35.314,156.655
C03124=1043.267,-27.327,422.401,169.548,35.312,156.655
C03125=1043.261,-27.576,422.414,169.546,35.312,156.655
C03126=1043.255,-27.825,422.427,169.544,35.311,156.655
C03127=1043.248,-28.075,422.442,169.542,35.310,156.655
C03128=1043.242,-28.324,422.456,169.540,35.309,156.654
C03129=1043.235,-28.574,422.469,169.538,35.308,156.654
C03130=1043.229,-28.824,422.482,169.536,35.308,156.654
C03131=1043.223,-29.073,422.496,169.534,35.307,156.654
C03132=1043.216,-29.323,422.509,169.532,35.305,156.654
C03133=1043.210,-29.572,422.523,169.530,35.305,156.654
C03134=1043.204,-29.821,422.536,169.528,35.304,156.654
C03135=1043.197,-30.071,422.549,169.524,35.303,156.654
C03136=1043.192,-30.322,422.563,169.522,35.302,156.653
C03137=1043.185,-30.571,422.576,169.520,35.301,156.653
C03138=1043.179,-30.821,422.590,169.518,35.301,156.653
C03139=1043.172,-31.070,422.603,169.516,35.299,156.653
C03140=1043.166,-31.319,422.616,169.514,35.299,156.653
C03141=1043.159,-31.569,422.630,169.512,35.298,156.653
C03142=1043.153,-31.818,422.643,169.510,35.297,156.653
C03143=1043.147,-32.068,422.656,169.508,35.296,156.653
C03144=1043.140,-32.318,422.670,169.506,35.295,156.652
C03145=1043.134,-32.567,422.683,169.504,35.294,156.652
C03146=1043.128,-32.817,422.697,169.502,35.294,156.652
C03147=1043.122,-33.067,422.711,169.500,35.292,156.652
C03148=1043.116,-33.316,422.723,169.498,35.292,156.652
C03149=1043.109,-33.566,422.736,169.495,35.291,156.652
C03150=1043.103,-33.815,422.750,169.493,35.290,156.652
C03151=1043.096,-34.065,422.763,169.491,35.289,156.652
C03152=1043.090,-34.314,422.777,169.489,35.288,156.651
C03153=1043.084,-34.563,422.790,169.487,35.287,156.651
C03154=1043.078,-34.813,422.802,169.485,35.287,156.651
C03155=1043.071,-35.094,422.818,169.483,35.285,156.651
C03156=1043.063,-35.375,422.833,169.480,35.285,156.651
C03157=1043.057,-35.656,422.847,169.477,35.283,156.651
C03158=1043.050,-35.937,422.863,169.475,35.283,156.651
C03159=1043.044,-36.187,422.876,169.473,35.282,156.651
C03160=1043.038,-36.436,422.889,169.471,35.281,156.650
C03161=1043.031,-36.686,422.903,169.468,35.280,156.650
C03162=1043.025,-36.935,422.916,169.466,35.279,156.650
C03163=1043.019,-37.185,422.928,169.464,35.278,156.650
C03164=1043.012,-37.435,422.942,169.462,35.278,156.650
C03165=1043.006,-37.684,422.955,169.460,35.276,156.650
C03166=1043.000,-37.933,422.968,169.458,35.276,156.650
C03167=1042.994,-38.184,422.981,169.456,35.275,156.650
C03168=1042.987,-38.433,422.994,169.454,35.274,156.649
C03169=1042.981,-38.682,423.008,169.452,35.273,156.649
C03170=1042.975,-38.932,423.020,169.450,35.272,156.649
C03171=1042.969,-39.181,423.034,169.447,35.272,156.649
C03172=1042.962,-39.431,423.047,169.445,35.271,156.649
C03173=1042.956,-39.681,423.060,169.443,35.270,156.649
C03174=1042.949,-39.930,423.072,169.441,35.269,156.649
C03175=1042.943,-40.180,423.085,169.439,35.269,156.649
C03176=1042.937,-40.429,423.098,169.437,35.268,156.649
C03177=1042.930,-40.679,423.112,169.435,35.267,156.648
C03178=1042.924,-40.929,423.124,169.433,35.267,156.648
C03179=1042.918,-41.178,423.137,169.430,35.266,156.648
C03180=1042.912,-41.428,423.150,169.428,35.265,156.648
C03181=1042.905,-41.677,423.163,169.425,35.264,156.648
C03182=1042.900,-41.927,423.175,169.423,35.263,156.648
C03183=1042.893,-42.177,423.189,169.421,35.262,156.648
C03184=1042.886,-42.426,423.202,169.419,35.262,156.648
C03185=1042.880,-42.676,423.214,169.417,35.261,156.648
C03186=1042.874,-42.925,423.228,169.414,35.260,156.647
C03187=1042.868,-43.175,423.240,169.412,35.260,156.647
C03188=1042.861,-43.424,423.253,169.410,35.259,156.647
C03189=1042.855,-43.674,423.265,169.408,35.258,156.647
C03190=1042.849,-43.923,423.279,169.406,35.257,156.647
C03191=1042.842,-44.174,423.292,169.404,35.257,156.647
C03192=1042.836,-44.423,423.305,169.402,35.256,156.647
C03193=1042.829,-44.673,423.317,169.399,35.255,156.647
C03194=1042.823,-44.922,423.329,169.397,35.255,156.647
C03195=1042.817,-45.172,423.343,169.395,35.254,156.647
C03196=1042.811,-45.422,423.355,169.393,35.253,156.647
C03197=1042.805,-45.671,423.368,169.391,35.253,156.646
C03198=1042.798,-45.920,423.380,169.389,35.252,156.646
C03199=1042.792,-46.170,423.394,169.386,35.251,156.646
C03200=1042.786,-46.420,423.406,169.384,35.250,156.646
C03201=1042.780,-46.669,423.419,169.382,35.250,156.646
C03202=1042.773,-46.918,423.431,169.380,35.249,156.646
C03203=1042.767,-47.168,423.444,169.378,35.248,156.646
C03204=1042.761,-47.418,423.457,169.376,35.248,156.646
C03205=1042.755,-47.667,423.470,169.374,35.247,156.646
C03206=1042.749,-47.917,423.482,169.371,35.246,156.646
C03207=1042.742,-48.166,423.495,169.369,35.245,156.645
C03208=1042.736,-48.417,423.508,169.367,35.245,156.645
C03209=1042.730,-48.667,423.521,169.364,35.243,156.645
C03210=1042.723,-48.916,423.533,169.362,35.243,156.645
C03211=1042.717,-49.166,423.546,169.360,35.242,156.645
C03212=1042.712,-49.415,423.558,169.357,35.241,156.645
C03213=1042.706,-49.664,423.571,169.355,35.240,156.645
C03214=1042.699,-49.914,423.583,169.353,35.240,156.645
C03215=1042.693,-50.164,423.596,169.351,35.239,156.645
C03216=1042.687,-50.413,423.608,169.349,35.238,156.644
C03217=1042.680,-50.663,423.621,169.346,35.238,156.645
C03218=1042.674,-50.913,423.634,169.344,35.238,156.644
C03219=1042.667,-51.194,423.647,169.342,35.237,156.644
C03220=1042.659,-51.475,423.661,169.339,35.236,156.644
C03221=1042.652,-51.757,423.676,169.337,35.235,156.644
C03222=1042.645,-52.038,423.689,169.334,35.235,156.644
C03223=1042.639,-52.288,423.701,169.332,35.235,156.644
C03224=1042.633,-52.538,423.713,169.330,35.234,156.644
C03225=1042.625,-52.787,423.726,169.328,35.233,156.644
C03226=1042.619,-53.037,423.738,169.325,35.232,156.644
C03227=1042.613,-53.286,423.751,169.323,35.232,156.644
C03228=1042.607,-53.536,423.763,169.321,35.232,156.644
C03229=1042.601,-53.785,423.775,169.319,35.231,156.644
C03230=1042.594,-54.035,423.787,169.316,35.230,156.644
C03231=1042.588,-54.285,423.799,169.314,35.230,156.644
C03232=1042.582,-54.534,423.812,169.312,35.229,156.643
C03233=1042.575,-54.784,423.824,169.310,35.229,156.643
C03234=1042.569,-55.034,423.836,169.308,35.228,156.643
C03235=1042.562,-55.283,423.849,169.305,35.228,156.643
C03236=1042.555,-55.532,423.861,169.303,35.227,156.643
C03237=1042.550,-55.782,423.873,169.301,35.226,156.643
C03238=1042.543,-56.032,423.885,169.299,35.226,156.643
C03239=1042.536,-56.281,423.897,169.296,35.226,156.643
C03240=1042.530,-56.531,423.910,169.294,35.225,156.643
C03241=1042.524,-56.781,423.922,169.292,35.224,156.643
C03242=1042.517,-57.031,423.934,169.290,35.224,156.643
C03243=1042.511,-57.280,423.946,169.287,35.223,156.643
C03244=1042.504,-57.530,423.958,169.285,35.223,156.643
C03245=1042.499,-57.779,423.970,169.283,35.222,156.643
C03246=1042.493,-58.029,423.982,169.281,35.222,156.643
C03247=1042.486,-58.278,423.994,169.278,35.221,156.642
C03248=1042.480,-58.529,424.006,169.276,35.220,156.642
C03249=1042.474,-58.778,424.018,169.274,35.220,156.642
C03250=1042.467,-59.028,424.030,169.272,35.220,156.642
C03251=1042.461,-59.278,424.043,169.269,35.219,156.642
C03252=1042.454,-59.527,424.055,169.266,35.218,156.642
C03253=1042.448,-59.776,424.066,169.264,35.218,156.642
C03254=1042.442,-60.026,424.079,169.262,35.217,156.642
C03255=1042.436,-60.276,424.091,169.260,35.217,156.642
C03256=1042.429,-60.525,424.103,169.257,35.217,156.642
C03257=1042.423,-60.775,424.115,169.255,35.216,156.642
C03258=1042.417,-61.025,424.127,169.253,35.215,156.642
C03259=1042.411,-61.274,424.138,169.251,35.215,156.642
C03260=1042.405,-61.524,424.151,169.248,35.214,156.642
C03261=1042.398,-61.774,424.162,169.246,35.214,156.642
C03262=1042.392,-62.023,424.174,169.244,35.213,156.641
C03263=1042.386,-62.273,424.187,169.241,35.213,156.642
C03264=1042.380,-62.522,424.199,169.239,35.212,156.641
C03265=1042.373,-62.772,424.210,169.237,35.212,156.641
C03266=1042.367,-63.022,424.222,169.235,35.211,156.641
C03267=1042.361,-63.272,424.234,169.232,35.211,156.641
C03268=1042.355,-63.521,424.246,169.230,35.210,156.641
C03269=1042.348,-63.770,424.258,169.228,35.210,156.641
C03270=1042.343,-64.021,424.270,169.226,35.209,156.641
C03271=1042.336,-64.270,424.282,169.223,35.208,156.641
C03272=1042.330,-64.519,424.293,169.221,35.208,156.641
C03273=1042.324,-64.769,424.306,169.219,35.208,156.641
C03274=1042.318,-65.019,424.317,169.217,35.207,156.641
C03275=1042.311,-65.269,424.329,169.214,35.207,156.641
C03276=1042.305,-65.518,424.341,169.212,35.206,156.641
C03277=1042.299,-65.768,424.352,169.210,35.205,156.641
C03278=1042.293,-66.018,424.364,169.207,35.205,156.641
C03279=1042.287,-66.267,424.376,169.205,35.205,156.641
C03280=1042.281,-66.516,424.389,169.203,35.205,156.641
C03281=1042.274,-66.767,424.400,169.201,35.204,156.640
C03282=1042.268,-67.016,424.412,169.198,35.203,156.640
C03283=1042.261,-67.299,424.425,169.196,35.203,156.640
C03284=1042.254,-67.582,424.438,169.193,35.202,156.640
C03285=1042.247,-67.864,424.452,169.191,35.202,156.640
C03286=1042.240,-68.147,424.465,169.188,35.201,156.640
C03287=1042.234,-68.396,424.476,169.186,35.201,156.640
C03288=1042.228,-68.646,424.488,169.184,35.200,156.640
C03289=1042.222,-68.895,424.500,169.181,35.200,156.640
C03290=1042.216,-69.145,424.511,169.179,35.199,156.640
C03291=1042.209,-69.395,424.523,169.177,35.199,156.640
C03292=1042.204,-69.644,424.535,169.174,35.198,156.640
C03293=1042.198,-69.894,424.547,169.172,35.198,156.640
C03294=1042.191,-70.144,424.558,169.170,35.198,156.640
C03295=1042.185,-70.393,424.569,169.168,35.197,156.640
C03296=1042.179,-70.643,424.582,169.165,35.196,156.640
C03297=1042.173,-70.893,424.593,169.163,35.196,156.640
C03298=1042.167,-71.142,424.605,169.161,35.195,156.640
C03299=1042.161,-71.393,424.616,169.158,35.195,156.640
C03300=1042.155,-71.642,424.628,169.156,35.195,156.640
C03301=1042.149,-71.892,424.639,169.154,35.195,156.640
C03302=1042.143,-72.141,424.651,169.152,35.194,156.639
C03303=1042.136,-72.391,424.662,169.149,35.193,156.639
C03304=1042.131,-72.640,424.674,169.147,35.193,156.639
C03305=1042.125,-72.890,424.686,169.145,35.192,156.639
C03306=1042.118,-73.140,424.698,169.142,35.192,156.639
C03307=1042.112,-73.389,424.709,169.140,35.191,156.639
C03308=1042.106,-73.639,424.720,169.138,35.191,156.639
C03309=1042.101,-73.889,424.732,169.135,35.191,156.639
C03310=1042.094,-74.138,424.744,169.133,35.191,156.639
C03311=1042.088,-74.388,424.755,169.131,35.190,156.639
C03312=1042.082,-74.638,424.766,169.128,35.190,156.639
C03313=1042.075,-74.888,424.778,169.126,35.189,156.639
C03314=1042.070,-75.137,424.789,169.124,35.189,156.639
C03315=1042.063,-75.387,424.800,169.121,35.189,156.639
C03316=1042.057,-75.636,424.812,169.119,35.188,156.639
C03317=1042.051,-75.886,424.823,169.117,35.188,156.639
C03318=1042.044,-76.136,424.833,169.114,35.188,156.639
C03319=1042.038,-76.385,424.845,169.112,35.187,156.639
C03320=1042.031,-76.635,424.856,169.110,35.187,156.639
C03321=1042.026,-76.885,424.867,169.107,35.187,156.639
C03322=1042.019,-77.134,424.879,169.105,35.186,156.639
C03323=1042.013,-77.384,424.890,169.103,35.186,156.639
C03324=1042.007,-77.634,424.901,169.100,35.186,156.639
C03325=1042.001,-77.884,424.912,169.098,35.185,156.639
C03326=1041.995,-78.133,424.924,169.096,35.185,156.639
C03327=1041.989,-78.383,424.935,169.093,35.185,156.639
C03328=1041.983,-78.633,424.946,169.091,35.185,156.639
C03329=1041.977,-78.882,424.957,169.089,35.185,156.639
C03330=1041.970,-79.132,424.969,169.086,35.184,156.639
C03331=1041.964,-79.381,424.980,169.084,35.184,156.639
C03332=1041.958,-79.632,424.991,169.082,35.184,156.639
C03333=1041.952,-79.881,425.002,169.079,35.184,156.639
C03334=1041.945,-80.131,425.013,169.077,35.183,156.639
C03335=1041.940,-80.380,425.024,169.075,35.183,156.639
C03336=1041.933,-80.630,425.036,169.072,35.183,156.639
C03337=1041.926,-80.879,425.046,169.070,35.183,156.639
C03338=1041.920,-81.129,425.057,169.067,35.182,156.639
C03339=1041.914,-81.379,425.068,169.065,35.182,156.639
C03340=1041.908,-81.629,425.079,169.063,35.182,156.639
C03341=1041.902,-81.878,425.090,169.060,35.182,156.639
C03342=1041.895,-82.128,425.101,169.058,35.181,156.639
C03343=1041.889,-82.378,425.112,169.055,35.181,156.639
C03344=1041.882,-82.628,425.122,169.053,35.181,156.639
C03345=1041.877,-82.877,425.133,169.051,35.181,156.639
C03346=1041.871,-83.127,425.144,169.048,35.181,156.639
C03347=1041.863,-83.411,425.157,169.046,35.180,156.639
C03348=1041.856,-83.697,425.169,169.043,35.180,156.639
C03349=1041.849,-83.981,425.181,169.040,35.180,156.639
C03350=1041.842,-84.266,425.194,169.037,35.180,156.639
C03351=1041.836,-84.516,425.205,169.035,35.180,156.639
C03352=1041.829,-84.766,425.216,169.033,35.180,156.639
C03353=1041.823,-85.015,425.227,169.030,35.180,156.639
C03354=1041.817,-85.265,425.238,169.028,35.180,156.639
C03355=1041.810,-85.514,425.248,169.025,35.180,156.639
C03356=1041.804,-85.764,425.259,169.023,35.179,156.639
C03357=1041.798,-86.014,425.270,169.021,35.179,156.639
C03358=1041.792,-86.264,425.280,169.018,35.179,156.639
C03359=1041.786,-86.513,425.291,169.016,35.179,156.639
C03360=1041.780,-86.764,425.302,169.013,35.179,156.639
C03361=1041.773,-87.013,425.312,169.011,35.179,156.639
C03362=1041.768,-87.262,425.323,169.009,35.178,156.639
C03363=1041.761,-87.512,425.335,169.006,35.178,156.639
C03364=1041.755,-87.762,425.345,169.004,35.178,156.639
C03365=1041.749,-88.011,425.356,169.001,35.178,156.639
C03366=1041.742,-88.261,425.366,168.999,35.178,156.639
C03367=1041.736,-88.510,425.377,168.997,35.178,156.639
C03368=1041.731,-88.761,425.387,168.994,35.178,156.639
C03369=1041.724,-89.010,425.398,168.992,35.178,156.639
C03370=1041.718,-89.260,425.409,168.989,35.178,156.639
C03371=1041.712,-89.509,425.420,168.987,35.177,156.639
C03372=1041.705,-89.759,425.430,168.985,35.177,156.639
C03373=1041.699,-90.009,425.441,168.982,35.177,156.639
C03374=1041.694,-90.259,425.451,168.980,35.177,156.639
C03375=1041.687,-90.509,425.462,168.977,35.177,156.639
C03376=1041.681,-90.758,425.473,168.975,35.177,156.639
C03377=1041.675,-91.007,425.483,168.972,35.177,156.639
C03378=1041.669,-91.257,425.494,168.970,35.176,156.639
C03379=1041.663,-91.508,425.505,168.968,35.176,156.639
C03380=1041.656,-91.757,425.515,168.965,35.176,156.639
C03381=1041.651,-92.006,425.526,168.963,35.176,156.639
C03382=1041.644,-92.256,425.536,168.960,35.176,156.639
C03383=1041.638,-92.506,425.547,168.958,35.176,156.639
C03384=1041.632,-92.756,425.558,168.956,35.176,156.639
C03385=1041.626,-93.005,425.568,168.953,35.176,156.639
C03386=1041.620,-93.255,425.579,168.951,35.176,156.639
C03387=1041.613,-93.505,425.589,168.948,35.176,156.639
C03388=1041.608,-93.755,425.600,168.946,35.176,156.639
C03389=1041.602,-94.004,425.610,168.943,35.176,156.639
C03390=1041.596,-94.254,425.620,168.941,35.175,156.639
C03391=1041.590,-94.503,425.631,168.939,35.175,156.639
C03392=1041.583,-94.753,425.641,168.936,35.175,156.639
C03393=1041.578,-95.003,425.652,168.934,35.175,156.639
C03394=1041.572,-95.253,425.663,168.931,35.175,156.639
C03395=1041.565,-95.502,425.673,168.929,35.175,156.639
C03396=1041.560,-95.752,425.683,168.927,35.175,156.639
C03397=1041.553,-96.001,425.693,168.924,35.175,156.640
C03398=1041.547,-96.252,425.704,168.922,35.175,156.640
C03399=1041.541,-96.501,425.714,168.919,35.175,156.640
C03400=1041.535,-96.751,425.725,168.917,35.175,156.640
C03401=1041.530,-97.001,425.735,168.914,35.175,156.640
C03402=1041.523,-97.250,425.745,168.912,35.175,156.640
C03403=1041.518,-97.500,425.756,168.910,35.175,156.640
C03404=1041.511,-97.749,425.766,168.907,35.175,156.640
C03405=1041.505,-98.000,425.776,168.905,35.175,156.640
C03406=1041.499,-98.249,425.787,168.902,35.175,156.640
C03407=1041.493,-98.499,425.796,168.900,35.175,156.640
C03408=1041.486,-98.748,425.806,168.897,35.175,156.640
C03409=1041.481,-98.998,425.817,168.895,35.175,156.640
C03410=1041.474,-99.248,425.827,168.893,35.176,156.640
C03411=1041.467,-99.535,425.838,168.890,35.176,156.640
C03412=1041.460,-99.822,425.851,168.888,35.175,156.640
C03413=1041.453,-100.109,425.862,168.885,35.175,156.640
C03414=1041.446,-100.397,425.873,168.882,35.176,156.640
C03415=1041.440,-100.646,425.884,168.879,35.176,156.640
C03416=1041.434,-100.896,425.894,168.877,35.176,156.640
C03417=1041.427,-101.146,425.903,168.875,35.176,156.640
C03418=1041.422,-101.395,425.914,168.872,35.176,156.640
C03419=1041.416,-101.645,425.924,168.870,35.176,156.640
C03420=1041.408,-101.895,425.934,168.867,35.176,156.640
C03421=1041.403,-102.145,425.944,168.865,35.177,156.641
C03422=1041.397,-102.395,425.954,168.862,35.176,156.641
C03423=1041.390,-102.644,425.964,168.860,35.176,156.641
C03424=1041.384,-102.894,425.974,168.857,35.177,156.641
C03425=1041.379,-103.144,425.984,168.855,35.177,156.641
C03426=1041.372,-103.393,425.994,168.852,35.177,156.641
C03427=1041.366,-103.643,426.004,168.850,35.177,156.641
C03428=1041.361,-103.893,426.014,168.847,35.177,156.641
C03429=1041.354,-104.142,426.024,168.845,35.177,156.641
C03430=1041.348,-104.392,426.034,168.842,35.178,156.641
C03431=1041.342,-104.642,426.043,168.840,35.178,156.641
C03432=1041.336,-104.891,426.054,168.837,35.178,156.641
C03433=1041.330,-105.141,426.064,168.835,35.178,156.641
C03434=1041.324,-105.391,426.073,168.832,35.178,156.641
C03435=1041.318,-105.641,426.083,168.830,35.178,156.641
C03436=1041.312,-105.890,426.094,168.828,35.179,156.641
C03437=1041.306,-106.140,426.103,168.825,35.178,156.641
C03438=1041.300,-106.390,426.113,168.823,35.178,156.642
C03439=1041.293,-106.639,426.123,168.820,35.179,156.642
C03440=1041.287,-106.889,426.132,168.818,35.179,156.642
C03441=1041.281,-107.139,426.143,168.815,35.179,156.642
C03442=1041.275,-107.388,426.153,168.813,35.179,156.642
C03443=1041.269,-107.638,426.162,168.810,35.180,156.642
C03444=1041.263,-107.888,426.172,168.808,35.180,156.642
C03445=1041.257,-108.138,426.181,168.805,35.180,156.642
C03446=1041.251,-108.388,426.191,168.804,35.180,156.642
C03447=1041.244,-108.637,426.201,168.801,35.180,156.642
C03448=1041.238,-108.887,426.211,168.799,35.181,156.642
C03449=1041.232,-109.137,426.221,168.796,35.181,156.642
C03450=1041.226,-109.387,426.230,168.794,35.181,156.642
C03451=1041.220,-109.636,426.240,168.791,35.182,156.643
C03452=1041.214,-109.886,426.250,168.789,35.182,156.643
C03453=1041.208,-110.136,426.259,168.786,35.182,156.643
C03454=1041.202,-110.386,426.269,168.784,35.182,156.643
C03455=1041.195,-110.636,426.278,168.781,35.183,156.643
C03456=1041.189,-110.885,426.288,168.779,35.183,156.643
C03457=1041.183,-111.135,426.297,168.776,35.183,156.643
C03458=1041.177,-111.385,426.307,168.773,35.183,156.643
C03459=1041.171,-111.634,426.316,168.771,35.184,156.643
C03460=1041.165,-111.884,426.326,168.768,35.184,156.643
C03461=1041.159,-112.133,426.336,168.766,35.184,156.643
C03462=1041.153,-112.383,426.346,168.763,35.184,156.643
C03463=1041.146,-112.633,426.355,168.761,35.185,156.643
C03464=1041.141,-112.883,426.365,168.758,35.185,156.644
C03465=1041.135,-113.133,426.374,168.756,35.185,156.644
C03466=1041.129,-113.383,426.384,168.753,35.186,156.644
C03467=1041.123,-113.633,426.393,168.751,35.186,156.644
C03468=1041.117,-113.882,426.403,168.748,35.186,156.644
C03469=1041.111,-114.132,426.412,168.746,35.186,156.644
C03470=1041.105,-114.381,426.422,168.743,35.187,156.644
C03471=1041.099,-114.631,426.431,168.741,35.187,156.644
C03472=1041.092,-114.881,426.441,168.738,35.187,156.644
C03473=1041.086,-115.131,426.450,168.737,35.188,156.644
C03474=1041.080,-115.381,426.460,168.734,35.188,156.644
C03475=1041.073,-115.666,426.470,168.731,35.189,156.645
C03476=1041.067,-115.953,426.481,168.728,35.189,156.645
C03477=1041.059,-116.238,426.492,168.725,35.189,156.645
C03478=1041.052,-116.525,426.503,168.723,35.190,156.645
C03479=1041.046,-116.775,426.512,168.720,35.190,156.645
C03480=1041.040,-117.025,426.521,168.718,35.190,156.645
C03481=1041.034,-117.274,426.530,168.715,35.191,156.645
C03482=1041.028,-117.524,426.540,168.712,35.191,156.645
C03483=1041.022,-117.774,426.549,168.710,35.191,156.645
C03484=1041.015,-118.023,426.558,168.707,35.192,156.645
C03485=1041.009,-118.274,426.567,168.705,35.192,156.646
C03486=1041.004,-118.523,426.576,168.702,35.193,156.646
C03487=1040.998,-118.773,426.586,168.700,35.193,156.646
C03488=1040.991,-119.023,426.595,168.697,35.193,156.646
C03489=1040.985,-119.272,426.605,168.695,35.194,156.646
C03490=1040.979,-119.523,426.614,168.692,35.195,156.646
C03491=1040.973,-119.772,426.623,168.690,35.194,156.646
C03492=1040.967,-120.021,426.632,168.687,35.195,156.646
C03493=1040.961,-120.272,426.641,168.684,35.196,156.646
C03494=1040.955,-120.522,426.651,168.682,35.196,156.647
C03495=1040.949,-120.771,426.660,168.680,35.197,156.647
C03496=1040.943,-121.021,426.669,168.678,35.197,156.647
C03497=1040.937,-121.271,426.678,168.675,35.197,156.647
C03498=1040.930,-121.520,426.687,168.673,35.198,156.647
C03499=1040.925,-121.770,426.696,168.670,35.198,156.647
C03500=1040.919,-122.020,426.705,168.668,35.199,156.647
C03501=1040.913,-122.270,426.715,168.665,35.199,156.647
C03502=1040.908,-122.519,426.723,168.663,35.199,156.647
C03503=1040.901,-122.769,426.732,168.660,35.200,156.648
C03504=1040.894,-123.019,426.742,168.657,35.200,156.648
C03505=1040.889,-123.269,426.751,168.655,35.201,156.648
C03506=1040.883,-123.518,426.760,168.652,35.202,156.648
C03507=1040.877,-123.768,426.769,168.650,35.202,156.648
C03508=1040.870,-124.018,426.778,168.647,35.203,156.648
C03509=1040.865,-124.267,426.787,168.645,35.203,156.648
C03510=1040.859,-124.518,426.796,168.642,35.203,156.648
C03511=1040.853,-124.767,426.805,168.640,35.204,156.648
C03512=1040.847,-125.017,426.813,168.637,35.204,156.649
C03513=1040.840,-125.267,426.823,168.634,35.205,156.649
C03514=1040.835,-125.517,426.832,168.632,35.205,156.649
C03515=1040.828,-125.766,426.840,168.630,35.206,156.649
C03516=1040.822,-126.016,426.849,168.628,35.207,156.649
C03517=1040.816,-126.266,426.859,168.625,35.207,156.649
C03518=1040.810,-126.515,426.866,168.623,35.208,156.649
C03519=1040.804,-126.765,426.876,168.620,35.208,156.650
C03520=1040.798,-127.016,426.885,168.617,35.209,156.650
C03521=1040.792,-127.264,426.893,168.615,35.209,156.650
C03522=1040.786,-127.515,426.902,168.612,35.210,156.650
C03523=1040.780,-127.764,426.912,168.610,35.211,156.650
C03524=1040.774,-128.014,426.921,168.607,35.211,156.650
C03525=1040.770,-128.264,426.930,168.605,35.210,156.650
C03526=1040.766,-128.514,426.941,168.603,35.210,156.650
C03527=1040.763,-128.763,426.951,168.601,35.209,156.650
C03528=1040.761,-129.014,426.963,168.599,35.208,156.650
C03529=1040.759,-129.263,426.976,168.597,35.206,156.649
C03530=1040.759,-129.513,426.988,168.595,35.203,156.649
C03531=1040.759,-129.763,427.002,168.593,35.200,156.649
C03532=1040.760,-130.014,427.016,168.591,35.196,156.648
C03533=1040.762,-130.264,427.030,168.590,35.193,156.647
C03534=1040.765,-130.513,427.046,168.589,35.188,156.647
C03535=1040.768,-130.764,427.062,168.587,35.184,156.646
C03536=1040.772,-131.014,427.078,168.586,35.178,156.645
C03537=1040.778,-131.264,427.095,168.586,35.173,156.644
C03538=1040.784,-131.514,427.113,168.584,35.167,156.643
C03539=1040.437,-131.538,426.855,168.538,35.361,156.676
C03540=1040.431,-131.289,426.837,168.538,35.368,156.678
C03541=1040.425,-131.039,426.820,168.539,35.373,156.678
C03542=1040.421,-130.788,426.804,168.541,35.378,156.679
C03543=1040.418,-130.537,426.788,168.542,35.383,156.680
C03544=1040.415,-130.288,426.772,168.543,35.387,156.681
C03545=1040.413,-130.038,426.758,168.545,35.391,156.682
C03546=1040.413,-129.788,426.743,168.546,35.395,156.682
C03547=1040.412,-129.537,426.730,168.548,35.398,156.683
C03548=1040.412,-129.288,426.717,168.549,35.400,156.683
C03549=1040.414,-129.037,426.705,168.551,35.402,156.683
C03550=1040.416,-128.788,426.694,168.553,35.403,156.683
C03551=1040.419,-128.537,426.683,168.555,35.405,156.684
C03552=1040.423,-128.287,426.672,168.557,35.405,156.684
C03553=1040.427,-128.038,426.662,168.560,35.406,156.684
C03554=1040.433,-127.788,426.653,168.562,35.406,156.684
C03555=1040.439,-127.539,426.644,168.565,35.405,156.684
C03556=1040.444,-127.289,426.635,168.567,35.404,156.683
C03557=1040.451,-127.039,426.626,168.570,35.404,156.683
C03558=1040.457,-126.789,426.617,168.572,35.403,156.683
C03559=1040.462,-126.540,426.608,168.575,35.403,156.683
C03560=1040.469,-126.290,426.600,168.578,35.402,156.683
C03561=1040.475,-126.041,426.591,168.580,35.401,156.683
C03562=1040.480,-125.790,426.582,168.583,35.400,156.683
C03563=1040.487,-125.541,426.573,168.585,35.400,156.682
C03564=1040.493,-125.291,426.564,168.588,35.399,156.682
C03565=1040.499,-125.041,426.555,168.591,35.399,156.682
C03566=1040.505,-124.791,426.547,168.593,35.398,156.682
C03567=1040.511,-124.542,426.537,168.596,35.397,156.682
C03568=1040.517,-124.292,426.529,168.598,35.397,156.682
C03569=1040.524,-124.042,426.520,168.601,35.397,156.682
C03570=1040.530,-123.792,426.510,168.603,35.396,156.682
C03571=1040.535,-123.543,426.502,168.605,35.396,156.682
C03572=1040.541,-123.293,426.492,168.608,35.395,156.681
C03573=1040.547,-123.042,426.483,168.610,35.395,156.681
C03574=1040.554,-122.794,426.475,168.613,35.394,156.681
C03575=1040.560,-122.544,426.465,168.615,35.393,156.681
C03576=1040.566,-122.293,426.456,168.618,35.393,156.681
C03577=1040.571,-122.044,426.447,168.620,35.393,156.681
C03578=1040.577,-121.794,426.437,168.623,35.392,156.681
C03579=1040.584,-121.544,426.429,168.626,35.392,156.681
C03580=1040.590,-121.295,426.420,168.628,35.391,156.680
C03581=1040.596,-121.045,426.410,168.631,35.391,156.680
C03582=1040.602,-120.795,426.401,168.633,35.390,156.680
C03583=1040.608,-120.545,426.392,168.636,35.389,156.680
C03584=1040.614,-120.295,426.382,168.638,35.390,156.680
C03585=1040.620,-120.046,426.374,168.641,35.389,156.680
C03586=1040.626,-119.796,426.365,168.643,35.388,156.680
C03587=1040.632,-119.546,426.355,168.646,35.388,156.680
C03588=1040.638,-119.297,426.346,168.649,35.387,156.680
C03589=1040.644,-119.047,426.337,168.651,35.387,156.680
C03590=1040.650,-118.797,426.328,168.653,35.387,156.679
C03591=1040.656,-118.547,426.318,168.655,35.386,156.679
C03592=1040.663,-118.298,426.309,168.658,35.386,156.679
C03593=1040.668,-118.048,426.301,168.660,35.385,156.679
C03594=1040.674,-117.798,426.291,168.663,35.385,156.679
C03595=1040.681,-117.549,426.282,168.666,35.385,156.679
C03596=1040.687,-117.299,426.272,168.668,35.384,156.679
C03597=1040.693,-117.049,426.262,168.671,35.383,156.679
C03598=1040.698,-116.799,426.254,168.673,35.383,156.679
C03599=1040.704,-116.549,426.244,168.676,35.383,156.678
C03600=1040.712,-116.263,426.234,168.679,35.382,156.678
C03601=1040.719,-115.977,426.222,168.682,35.382,156.678
C03602=1040.726,-115.691,426.212,168.684,35.381,156.678
C03603=1040.733,-115.404,426.201,168.687,35.381,156.678
C03604=1040.739,-115.155,426.192,168.690,35.381,156.678
C03605=1040.745,-114.905,426.183,168.692,35.380,156.678
C03606=1040.751,-114.656,426.173,168.695,35.380,156.678
C03607=1040.757,-114.406,426.163,168.698,35.380,156.678
C03608=1040.763,-114.156,426.154,168.700,35.379,156.678
C03609=1040.769,-113.906,426.145,168.703,35.378,156.677
C03610=1040.775,-113.656,426.135,168.705,35.379,156.677
C03611=1040.781,-113.406,426.126,168.708,35.378,156.677
C03612=1040.787,-113.157,426.117,168.710,35.378,156.677
C03613=1040.793,-112.907,426.107,168.712,35.377,156.677
C03614=1040.799,-112.657,426.098,168.714,35.377,156.677
C03615=1040.806,-112.407,426.088,168.717,35.377,156.677
C03616=1040.812,-112.158,426.078,168.719,35.376,156.677
C03617=1040.818,-111.908,426.069,168.722,35.376,156.677
C03618=1040.823,-111.658,426.059,168.724,35.376,156.677
C03619=1040.829,-111.408,426.049,168.727,35.375,156.677
C03620=1040.836,-111.158,426.040,168.729,35.375,156.677
C03621=1040.841,-110.909,426.030,168.732,35.375,156.676
C03622=1040.847,-110.659,426.021,168.734,35.375,156.676
C03623=1040.854,-110.409,426.011,168.737,35.374,156.676
C03624=1040.860,-110.160,426.001,168.740,35.374,156.676
C03625=1040.866,-109.911,425.991,168.742,35.374,156.676
C03626=1040.872,-109.661,425.982,168.745,35.373,156.676
C03627=1040.879,-109.411,425.972,168.747,35.373,156.676
C03628=1040.885,-109.161,425.963,168.750,35.373,156.676
C03629=1040.891,-108.911,425.953,168.752,35.373,156.676
C03630=1040.897,-108.662,425.944,168.755,35.372,156.676
C03631=1040.903,-108.412,425.934,168.757,35.372,156.676
